   S704_BT_CODE_2018.RBT14_STANDARD_WELD_DATA := W#16#0;
   S704_BT_CODE_2018.RBT15_STANDARD_WELD_DATA := W#16#0;
   S704_BT_CODE_2018.RBT16_STANDARD_WELD_DATA := W#16#0;
   S704_BT_CODE_2018.RBT17_STANDARD_WELD_DATA := W#16#0;
   S704_BT_CODE_2018.RBT18_STANDARD_WELD_DATA := W#16#0;
   S704_BT_CODE_2018.RBT19_STANDARD_WELD_DATA := W#16#0;
   S704_BT_CODE_2018.RBT20_STANDARD_WELD_DATA := W#16#0;
   S704_BT_CODE_2018.RBT21_STANDARD_WELD_DATA := W#16#0;
   S704_BT_CODE_2018.RBT22_STANDARD_WELD_DATA := W#16#0;
   S704_BT_CODE_2018.RBT23_STANDARD_WELD_DAT := W#16#0;
   S704_BT_CODE_2018.RBT24_STANDARD_WELD_DAT := W#16#0;
   S704_BT_CODE_2018.CHK_WORD := W#16#0;
   S704_BT_CODE_2018.TEST_TEMP[1] := B#16#0;
   S704_BT_CODE_2018.TEST_TEMP[2] := B#16#0;
   S704_BT_CODE_2018.TEST_TEMP[3] := B#16#0;
   S704_BT_CODE_2018.TEST_TEMP[4] := B#16#0;
   S704_BT_CODE_2018.TEST_TEMP[5] := B#16#0;
   S704_BT_CODE_2018.TEST_TEMP[6] := B#16#0;
   S704_BT_CODE_2018.TEST_TEMP[7] := B#16#0;
   S704_BT_CODE_2018.TEST_TEMP[8] := B#16#0;
   S704_BT_CODE_2018.TEST_TEMP[9] := B#16#0;
   S704_BT_CODE_2018.TEST_TEMP[10] := B#16#0;
   S704_BT_CODE_2018.TEST_TEMP[11] := B#16#0;
   S704_BT_CODE_2018.TEST_TEMP[12] := B#16#0;
   S704_BT_CODE_2018.TEST_TEMP[13] := B#16#0;
   S704_BT_CODE_2018.TEST_TEMP[14] := B#16#0;
   S704_BT_CODE_2018.TEST_TEMP[15] := B#16#0;
   S704_BT_CODE_2018.TEST_TEMP[16] := B#16#0;
   S704_BT_CODE_2018.TEST_TEMP[17] := B#16#0;
   S704_BT_CODE_2018.TEST_TEMP[18] := B#16#0;
   S704_BT_CODE_2018.TEST_TEMP[19] := B#16#0;
   S704_BT_CODE_2018.TEST_TEMP[20] := B#16#0;
   S704_BT_CODE_2018.TEST_TEMP[21] := B#16#0;
   S704_BT_CODE_2018.TEST_TEMP[22] := B#16#0;
   S704_BT_CODE_2018.TEST_TEMP[23] := B#16#0;
   S704_BT_CODE_2018.TEST_TEMP[24] := B#16#0;
   S704_BT_CODE_2018.TEST_TEMP[25] := B#16#0;
   S704_BT_CODE_2018.TEST_TEMP[26] := B#16#0;
   S704_BT_CODE_2018.TEST_TEMP[27] := B#16#0;
   S704_BT_CODE_2018.TEST_TEMP[28] := B#16#0;
   S704_BT_CODE_2018.TEST_TEMP[29] := B#16#0;
   S704_BT_CODE_2018.TEST_TEMP[30] := B#16#0;
   S704_BT_CODE_2018.TEST_TEMP[31] := B#16#0;
   S704_BT_CODE_2018.TEST_TEMP[32] := B#16#0;
   S704_BT_CODE_2018.TEST_TEMP[33] := B#16#0;
   S704_BT_CODE_2018.TEST_TEMP[34] := B#16#0;
   S704_BT_CODE_2018.TEST_TEMP[35] := B#16#0;
   S704_BT_CODE_2018.TEST_TEMP[36] := B#16#0;
   S704_BT_CODE_2018.TEST_TEMP[37] := B#16#0;
   S704_BT_CODE_2018.TEST_TEMP[38] := B#16#0;
   S704_BT_CODE_2018.TEST_TEMP[39] := B#16#0;
   S704_BT_CODE_2018.TEST_TEMP[40] := B#16#0;
   S704_BT_CODE_2019.STATION_MAIN := W#16#0;
   S704_BT_CODE_2019.DISTINCTION_LH_RH := W#16#0;
   S704_BT_CODE_2019.STAION_NUMBER := W#16#0;
   S704_BT_CODE_2019.BODY_TYPE_1ST := W#16#0;
   S704_BT_CODE_2019.BODY_TYPE_OPTION := W#16#0;
   S704_BT_CODE_2019.RBT1_STANDARD_WELD_DATA := W#16#0;
   S704_BT_CODE_2019.RBT2_STANDARD_WELD_DATA := W#16#0;
   S704_BT_CODE_2019.RBT3_STANDARD_WELD_DATA := W#16#0;
   S704_BT_CODE_2019.RBT4_STANDARD_WELD_DATA := W#16#0;
   S704_BT_CODE_2019.RBT5_STANDARD_WELD_DATA := W#16#0;
   S704_BT_CODE_2019.RBT6_STANDARD_WELD_DATA := W#16#0;
   S704_BT_CODE_2019.RBT7_STANDARD_WELD_DATA := W#16#0;
   S704_BT_CODE_2019.RBT8_STANDARD_WELD_DATA := W#16#0;
   S704_BT_CODE_2019.RBT9_STANDARD_WELD_DATA := W#16#0;
   S704_BT_CODE_2019.RBT10_STANDARD_WELD_DATA := W#16#0;
   S704_BT_CODE_2019.RBT11_STANDARD_WELD_DATA := W#16#0;
   S704_BT_CODE_2019.RBT12_STANDARD_WELD_DATA := W#16#0;
   S704_BT_CODE_2019.RBT13_STANDARD_WELD_DATA := W#16#0;
   S704_BT_CODE_2019.RBT14_STANDARD_WELD_DATA := W#16#0;
   S704_BT_CODE_2019.RBT15_STANDARD_WELD_DATA := W#16#0;
   S704_BT_CODE_2019.RBT16_STANDARD_WELD_DATA := W#16#0;
   S704_BT_CODE_2019.RBT17_STANDARD_WELD_DATA := W#16#0;
   S704_BT_CODE_2019.RBT18_STANDARD_WELD_DATA := W#16#0;
   S704_BT_CODE_2019.RBT19_STANDARD_WELD_DATA := W#16#0;
   S704_BT_CODE_2019.RBT20_STANDARD_WELD_DATA := W#16#0;
   S704_BT_CODE_2019.RBT21_STANDARD_WELD_DATA := W#16#0;
   S704_BT_CODE_2019.RBT22_STANDARD_WELD_DATA := W#16#0;
   S704_BT_CODE_2019.RBT23_STANDARD_WELD_DAT := W#16#0;
   S704_BT_CODE_2019.RBT24_STANDARD_WELD_DAT := W#16#0;
   S704_BT_CODE_2019.CHK_WORD := W#16#0;
   S704_BT_CODE_2019.TEST_TEMP[1] := B#16#0;
   S704_BT_CODE_2019.TEST_TEMP[2] := B#16#0;
   S704_BT_CODE_2019.TEST_TEMP[3] := B#16#0;
   S704_BT_CODE_2019.TEST_TEMP[4] := B#16#0;
   S704_BT_CODE_2019.TEST_TEMP[5] := B#16#0;
   S704_BT_CODE_2019.TEST_TEMP[6] := B#16#0;
   S704_BT_CODE_2019.TEST_TEMP[7] := B#16#0;
   S704_BT_CODE_2019.TEST_TEMP[8] := B#16#0;
   S704_BT_CODE_2019.TEST_TEMP[9] := B#16#0;
   S704_BT_CODE_2019.TEST_TEMP[10] := B#16#0;
   S704_BT_CODE_2019.TEST_TEMP[11] := B#16#0;
   S704_BT_CODE_2019.TEST_TEMP[12] := B#16#0;
   S704_BT_CODE_2019.TEST_TEMP[13] := B#16#0;
   S704_BT_CODE_2019.TEST_TEMP[14] := B#16#0;
   S704_BT_CODE_2019.TEST_TEMP[15] := B#16#0;
   S704_BT_CODE_2019.TEST_TEMP[16] := B#16#0;
   S704_BT_CODE_2019.TEST_TEMP[17] := B#16#0;
   S704_BT_CODE_2019.TEST_TEMP[18] := B#16#0;
   S704_BT_CODE_2019.TEST_TEMP[19] := B#16#0;
   S704_BT_CODE_2019.TEST_TEMP[20] := B#16#0;
   S704_BT_CODE_2019.TEST_TEMP[21] := B#16#0;
   S704_BT_CODE_2019.TEST_TEMP[22] := B#16#0;
   S704_BT_CODE_2019.TEST_TEMP[23] := B#16#0;
   S704_BT_CODE_2019.TEST_TEMP[24] := B#16#0;
   S704_BT_CODE_2019.TEST_TEMP[25] := B#16#0;
   S704_BT_CODE_2019.TEST_TEMP[26] := B#16#0;
   S704_BT_CODE_2019.TEST_TEMP[27] := B#16#0;
   S704_BT_CODE_2019.TEST_TEMP[28] := B#16#0;
   S704_BT_CODE_2019.TEST_TEMP[29] := B#16#0;
   S704_BT_CODE_2019.TEST_TEMP[30] := B#16#0;
   S704_BT_CODE_2019.TEST_TEMP[31] := B#16#0;
   S704_BT_CODE_2019.TEST_TEMP[32] := B#16#0;
   S704_BT_CODE_2019.TEST_TEMP[33] := B#16#0;
   S704_BT_CODE_2019.TEST_TEMP[34] := B#16#0;
   S704_BT_CODE_2019.TEST_TEMP[35] := B#16#0;
   S704_BT_CODE_2019.TEST_TEMP[36] := B#16#0;
   S704_BT_CODE_2019.TEST_TEMP[37] := B#16#0;
   S704_BT_CODE_2019.TEST_TEMP[38] := B#16#0;
   S704_BT_CODE_2019.TEST_TEMP[39] := B#16#0;
   S704_BT_CODE_2019.TEST_TEMP[40] := B#16#0;
   S704_BT_CODE_2020.STATION_MAIN := W#16#0;
   S704_BT_CODE_2020.DISTINCTION_LH_RH := W#16#0;
   S704_BT_CODE_2020.STAION_NUMBER := W#16#0;
   S704_BT_CODE_2020.BODY_TYPE_1ST := W#16#0;
   S704_BT_CODE_2020.BODY_TYPE_OPTION := W#16#0;
   S704_BT_CODE_2020.RBT1_STANDARD_WELD_DATA := W#16#0;
   S704_BT_CODE_2020.RBT2_STANDARD_WELD_DATA := W#16#0;
   S704_BT_CODE_2020.RBT3_STANDARD_WELD_DATA := W#16#0;
   S704_BT_CODE_2020.RBT4_STANDARD_WELD_DATA := W#16#0;
   S704_BT_CODE_2020.RBT5_STANDARD_WELD_DATA := W#16#0;
   S704_BT_CODE_2020.RBT6_STANDARD_WELD_DATA := W#16#0;
   S704_BT_CODE_2020.RBT7_STANDARD_WELD_DATA := W#16#0;
   S704_BT_CODE_2020.RBT8_STANDARD_WELD_DATA := W#16#0;
   S704_BT_CODE_2020.RBT9_STANDARD_WELD_DATA := W#16#0;
   S704_BT_CODE_2020.RBT10_STANDARD_WELD_DATA := W#16#0;
   S704_BT_CODE_2020.RBT11_STANDARD_WELD_DATA := W#16#0;
   S704_BT_CODE_2020.RBT12_STANDARD_WELD_DATA := W#16#0;
   S704_BT_CODE_2020.RBT13_STANDARD_WELD_DATA := W#16#0;
   S704_BT_CODE_2020.RBT14_STANDARD_WELD_DATA := W#16#0;
   S704_BT_CODE_2020.RBT15_STANDARD_WELD_DATA := W#16#0;
   S704_BT_CODE_2020.RBT16_STANDARD_WELD_DATA := W#16#0;
   S704_BT_CODE_2020.RBT17_STANDARD_WELD_DATA := W#16#0;
   S704_BT_CODE_2020.RBT18_STANDARD_WELD_DATA := W#16#0;
   S704_BT_CODE_2020.RBT19_STANDARD_WELD_DATA := W#16#0;
   S704_BT_CODE_2020.RBT20_STANDARD_WELD_DATA := W#16#0;
   S704_BT_CODE_2020.RBT21_STANDARD_WELD_DATA := W#16#0;
   S704_BT_CODE_2020.RBT22_STANDARD_WELD_DATA := W#16#0;
   S704_BT_CODE_2020.RBT23_STANDARD_WELD_DAT := W#16#0;
   S704_BT_CODE_2020.RBT24_STANDARD_WELD_DAT := W#16#0;
   S704_BT_CODE_2020.CHK_WORD := W#16#0;
   S704_BT_CODE_2020.TEST_TEMP[1] := B#16#0;
   S704_BT_CODE_2020.TEST_TEMP[2] := B#16#0;
   S704_BT_CODE_2020.TEST_TEMP[3] := B#16#0;
   S704_BT_CODE_2020.TEST_TEMP[4] := B#16#0;
   S704_BT_CODE_2020.TEST_TEMP[5] := B#16#0;
   S704_BT_CODE_2020.TEST_TEMP[6] := B#16#0;
   S704_BT_CODE_2020.TEST_TEMP[7] := B#16#0;
   S704_BT_CODE_2020.TEST_TEMP[8] := B#16#0;
   S704_BT_CODE_2020.TEST_TEMP[9] := B#16#0;
   S704_BT_CODE_2020.TEST_TEMP[10] := B#16#0;
   S704_BT_CODE_2020.TEST_TEMP[11] := B#16#0;
   S704_BT_CODE_2020.TEST_TEMP[12] := B#16#0;
   S704_BT_CODE_2020.TEST_TEMP[13] := B#16#0;
   S704_BT_CODE_2020.TEST_TEMP[14] := B#16#0;
   S704_BT_CODE_2020.TEST_TEMP[15] := B#16#0;
   S704_BT_CODE_2020.TEST_TEMP[16] := B#16#0;
   S704_BT_CODE_2020.TEST_TEMP[17] := B#16#0;
   S704_BT_CODE_2020.TEST_TEMP[18] := B#16#0;
   S704_BT_CODE_2020.TEST_TEMP[19] := B#16#0;
   S704_BT_CODE_2020.TEST_TEMP[20] := B#16#0;
   S704_BT_CODE_2020.TEST_TEMP[21] := B#16#0;
   S704_BT_CODE_2020.TEST_TEMP[22] := B#16#0;
   S704_BT_CODE_2020.TEST_TEMP[23] := B#16#0;
   S704_BT_CODE_2020.TEST_TEMP[24] := B#16#0;
   S704_BT_CODE_2020.TEST_TEMP[25] := B#16#0;
   S704_BT_CODE_2020.TEST_TEMP[26] := B#16#0;
   S704_BT_CODE_2020.TEST_TEMP[27] := B#16#0;
   S704_BT_CODE_2020.TEST_TEMP[28] := B#16#0;
   S704_BT_CODE_2020.TEST_TEMP[29] := B#16#0;
   S704_BT_CODE_2020.TEST_TEMP[30] := B#16#0;
   S704_BT_CODE_2020.TEST_TEMP[31] := B#16#0;
   S704_BT_CODE_2020.TEST_TEMP[32] := B#16#0;
   S704_BT_CODE_2020.TEST_TEMP[33] := B#16#0;
   S704_BT_CODE_2020.TEST_TEMP[34] := B#16#0;
   S704_BT_CODE_2020.TEST_TEMP[35] := B#16#0;
   S704_BT_CODE_2020.TEST_TEMP[36] := B#16#0;
   S704_BT_CODE_2020.TEST_TEMP[37] := B#16#0;
   S704_BT_CODE_2020.TEST_TEMP[38] := B#16#0;
   S704_BT_CODE_2020.TEST_TEMP[39] := B#16#0;
   S704_BT_CODE_2020.TEST_TEMP[40] := B#16#0;
   S704_BT_CODE_2021.STATION_MAIN := W#16#0;
   S704_BT_CODE_2021.DISTINCTION_LH_RH := W#16#0;
   S704_BT_CODE_2021.STAION_NUMBER := W#16#0;
   S704_BT_CODE_2021.BODY_TYPE_1ST := W#16#0;
   S704_BT_CODE_2021.BODY_TYPE_OPTION := W#16#0;
   S704_BT_CODE_2021.RBT1_STANDARD_WELD_DATA := W#16#0;
   S704_BT_CODE_2021.RBT2_STANDARD_WELD_DATA := W#16#0;
   S704_BT_CODE_2021.RBT3_STANDARD_WELD_DATA := W#16#0;
   S704_BT_CODE_2021.RBT4_STANDARD_WELD_DATA := W#16#0;
   S704_BT_CODE_2021.RBT5_STANDARD_WELD_DATA := W#16#0;
   S704_BT_CODE_2021.RBT6_STANDARD_WELD_DATA := W#16#0;
   S704_BT_CODE_2021.RBT7_STANDARD_WELD_DATA := W#16#0;
   S704_BT_CODE_2021.RBT8_STANDARD_WELD_DATA := W#16#0;
   S704_BT_CODE_2021.RBT9_STANDARD_WELD_DATA := W#16#0;
   S704_BT_CODE_2021.RBT10_STANDARD_WELD_DATA := W#16#0;
   S704_BT_CODE_2021.RBT11_STANDARD_WELD_DATA := W#16#0;
   S704_BT_CODE_2021.RBT12_STANDARD_WELD_DATA := W#16#0;
   S704_BT_CODE_2021.RBT13_STANDARD_WELD_DATA := W#16#0;
   S704_BT_CODE_2021.RBT14_STANDARD_WELD_DATA := W#16#0;
   S704_BT_CODE_2021.RBT15_STANDARD_WELD_DATA := W#16#0;
   S704_BT_CODE_2021.RBT16_STANDARD_WELD_DATA := W#16#0;
   S704_BT_CODE_2021.RBT17_STANDARD_WELD_DATA := W#16#0;
   S704_BT_CODE_2021.RBT18_STANDARD_WELD_DATA := W#16#0;
   S704_BT_CODE_2021.RBT19_STANDARD_WELD_DATA := W#16#0;
   S704_BT_CODE_2021.RBT20_STANDARD_WELD_DATA := W#16#0;
   S704_BT_CODE_2021.RBT21_STANDARD_WELD_DATA := W#16#0;
   S704_BT_CODE_2021.RBT22_STANDARD_WELD_DATA := W#16#0;
   S704_BT_CODE_2021.RBT23_STANDARD_WELD_DAT := W#16#0;
   S704_BT_CODE_2021.RBT24_STANDARD_WELD_DAT := W#16#0;
   S704_BT_CODE_2021.CHK_WORD := W#16#0;
   S704_BT_CODE_2021.TEST_TEMP[1] := B#16#0;
   S704_BT_CODE_2021.TEST_TEMP[2] := B#16#0;
   S704_BT_CODE_2021.TEST_TEMP[3] := B#16#0;
   S704_BT_CODE_2021.TEST_TEMP[4] := B#16#0;
   S704_BT_CODE_2021.TEST_TEMP[5] := B#16#0;
   S704_BT_CODE_2021.TEST_TEMP[6] := B#16#0;
   S704_BT_CODE_2021.TEST_TEMP[7] := B#16#0;
   S704_BT_CODE_2021.TEST_TEMP[8] := B#16#0;
   S704_BT_CODE_2021.TEST_TEMP[9] := B#16#0;
   S704_BT_CODE_2021.TEST_TEMP[10] := B#16#0;
   S704_BT_CODE_2021.TEST_TEMP[11] := B#16#0;
   S704_BT_CODE_2021.TEST_TEMP[12] := B#16#0;
   S704_BT_CODE_2021.TEST_TEMP[13] := B#16#0;
   S704_BT_CODE_2021.TEST_TEMP[14] := B#16#0;
   S704_BT_CODE_2021.TEST_TEMP[15] := B#16#0;
   S704_BT_CODE_2021.TEST_TEMP[16] := B#16#0;
   S704_BT_CODE_2021.TEST_TEMP[17] := B#16#0;
   S704_BT_CODE_2021.TEST_TEMP[18] := B#16#0;
   S704_BT_CODE_2021.TEST_TEMP[19] := B#16#0;
   S704_BT_CODE_2021.TEST_TEMP[20] := B#16#0;
   S704_BT_CODE_2021.TEST_TEMP[21] := B#16#0;
   S704_BT_CODE_2021.TEST_TEMP[22] := B#16#0;
   S704_BT_CODE_2021.TEST_TEMP[23] := B#16#0;
   S704_BT_CODE_2021.TEST_TEMP[24] := B#16#0;
   S704_BT_CODE_2021.TEST_TEMP[25] := B#16#0;
   S704_BT_CODE_2021.TEST_TEMP[26] := B#16#0;
   S704_BT_CODE_2021.TEST_TEMP[27] := B#16#0;
   S704_BT_CODE_2021.TEST_TEMP[28] := B#16#0;
   S704_BT_CODE_2021.TEST_TEMP[29] := B#16#0;
   S704_BT_CODE_2021.TEST_TEMP[30] := B#16#0;
   S704_BT_CODE_2021.TEST_TEMP[31] := B#16#0;
   S704_BT_CODE_2021.TEST_TEMP[32] := B#16#0;
   S704_BT_CODE_2021.TEST_TEMP[33] := B#16#0;
   S704_BT_CODE_2021.TEST_TEMP[34] := B#16#0;
   S704_BT_CODE_2021.TEST_TEMP[35] := B#16#0;
   S704_BT_CODE_2021.TEST_TEMP[36] := B#16#0;
   S704_BT_CODE_2021.TEST_TEMP[37] := B#16#0;
   S704_BT_CODE_2021.TEST_TEMP[38] := B#16#0;
   S704_BT_CODE_2021.TEST_TEMP[39] := B#16#0;
   S704_BT_CODE_2021.TEST_TEMP[40] := B#16#0;
   S704_BT_CODE_2022.STATION_MAIN := W#16#0;
   S704_BT_CODE_2022.DISTINCTION_LH_RH := W#16#0;
   S704_BT_CODE_2022.STAION_NUMBER := W#16#0;
   S704_BT_CODE_2022.BODY_TYPE_1ST := W#16#0;
   S704_BT_CODE_2022.BODY_TYPE_OPTION := W#16#0;
   S704_BT_CODE_2022.RBT1_STANDARD_WELD_DATA := W#16#0;
   S704_BT_CODE_2022.RBT2_STANDARD_WELD_DATA := W#16#0;
   S704_BT_CODE_2022.RBT3_STANDARD_WELD_DATA := W#16#0;
   S704_BT_CODE_2022.RBT4_STANDARD_WELD_DATA := W#16#0;
   S704_BT_CODE_2022.RBT5_STANDARD_WELD_DATA := W#16#0;
   S704_BT_CODE_2022.RBT6_STANDARD_WELD_DATA := W#16#0;
   S704_BT_CODE_2022.RBT7_STANDARD_WELD_DATA := W#16#0;
   S704_BT_CODE_2022.RBT8_STANDARD_WELD_DATA := W#16#0;
   S704_BT_CODE_2022.RBT9_STANDARD_WELD_DATA := W#16#0;
   S704_BT_CODE_2022.RBT10_STANDARD_WELD_DATA := W#16#0;
   S704_BT_CODE_2022.RBT11_STANDARD_WELD_DATA := W#16#0;
   S704_BT_CODE_2022.RBT12_STANDARD_WELD_DATA := W#16#0;
   S704_BT_CODE_2022.RBT13_STANDARD_WELD_DATA := W#16#0;
   S704_BT_CODE_2022.RBT14_STANDARD_WELD_DATA := W#16#0;
   S704_BT_CODE_2022.RBT15_STANDARD_WELD_DATA := W#16#0;
   S704_BT_CODE_2022.RBT16_STANDARD_WELD_DATA := W#16#0;
   S704_BT_CODE_2022.RBT17_STANDARD_WELD_DATA := W#16#0;
   S704_BT_CODE_2022.RBT18_STANDARD_WELD_DATA := W#16#0;
   S704_BT_CODE_2022.RBT19_STANDARD_WELD_DATA := W#16#0;
   S704_BT_CODE_2022.RBT20_STANDARD_WELD_DATA := W#16#0;
   S704_BT_CODE_2022.RBT21_STANDARD_WELD_DATA := W#16#0;
   S704_BT_CODE_2022.RBT22_STANDARD_WELD_DATA := W#16#0;
   S704_BT_CODE_2022.RBT23_STANDARD_WELD_DAT := W#16#0;
   S704_BT_CODE_2022.RBT24_STANDARD_WELD_DAT := W#16#0;
   S704_BT_CODE_2022.CHK_WORD := W#16#0;
   S704_BT_CODE_2022.TEST_TEMP[1] := B#16#0;
   S704_BT_CODE_2022.TEST_TEMP[2] := B#16#0;
   S704_BT_CODE_2022.TEST_TEMP[3] := B#16#0;
   S704_BT_CODE_2022.TEST_TEMP[4] := B#16#0;
   S704_BT_CODE_2022.TEST_TEMP[5] := B#16#0;
   S704_BT_CODE_2022.TEST_TEMP[6] := B#16#0;
   S704_BT_CODE_2022.TEST_TEMP[7] := B#16#0;
   S704_BT_CODE_2022.TEST_TEMP[8] := B#16#0;
   S704_BT_CODE_2022.TEST_TEMP[9] := B#16#0;
   S704_BT_CODE_2022.TEST_TEMP[10] := B#16#0;
   S704_BT_CODE_2022.TEST_TEMP[11] := B#16#0;
   S704_BT_CODE_2022.TEST_TEMP[12] := B#16#0;
   S704_BT_CODE_2022.TEST_TEMP[13] := B#16#0;
   S704_BT_CODE_2022.TEST_TEMP[14] := B#16#0;
   S704_BT_CODE_2022.TEST_TEMP[15] := B#16#0;
   S704_BT_CODE_2022.TEST_TEMP[16] := B#16#0;
   S704_BT_CODE_2022.TEST_TEMP[17] := B#16#0;
   S704_BT_CODE_2022.TEST_TEMP[18] := B#16#0;
   S704_BT_CODE_2022.TEST_TEMP[19] := B#16#0;
   S704_BT_CODE_2022.TEST_TEMP[20] := B#16#0;
   S704_BT_CODE_2022.TEST_TEMP[21] := B#16#0;
   S704_BT_CODE_2022.TEST_TEMP[22] := B#16#0;
   S704_BT_CODE_2022.TEST_TEMP[23] := B#16#0;
   S704_BT_CODE_2022.TEST_TEMP[24] := B#16#0;
   S704_BT_CODE_2022.TEST_TEMP[25] := B#16#0;
   S704_BT_CODE_2022.TEST_TEMP[26] := B#16#0;
   S704_BT_CODE_2022.TEST_TEMP[27] := B#16#0;
   S704_BT_CODE_2022.TEST_TEMP[28] := B#16#0;
   S704_BT_CODE_2022.TEST_TEMP[29] := B#16#0;
   S704_BT_CODE_2022.TEST_TEMP[30] := B#16#0;
   S704_BT_CODE_2022.TEST_TEMP[31] := B#16#0;
   S704_BT_CODE_2022.TEST_TEMP[32] := B#16#0;
   S704_BT_CODE_2022.TEST_TEMP[33] := B#16#0;
   S704_BT_CODE_2022.TEST_TEMP[34] := B#16#0;
   S704_BT_CODE_2022.TEST_TEMP[35] := B#16#0;
   S704_BT_CODE_2022.TEST_TEMP[36] := B#16#0;
   S704_BT_CODE_2022.TEST_TEMP[37] := B#16#0;
   S704_BT_CODE_2022.TEST_TEMP[38] := B#16#0;
   S704_BT_CODE_2022.TEST_TEMP[39] := B#16#0;
   S704_BT_CODE_2022.TEST_TEMP[40] := B#16#0;
   S704_BT_CODE_2023.STATION_MAIN := W#16#0;
   S704_BT_CODE_2023.DISTINCTION_LH_RH := W#16#0;
   S704_BT_CODE_2023.STAION_NUMBER := W#16#0;
   S704_BT_CODE_2023.BODY_TYPE_1ST := W#16#0;
   S704_BT_CODE_2023.BODY_TYPE_OPTION := W#16#0;
   S704_BT_CODE_2023.RBT1_STANDARD_WELD_DATA := W#16#0;
   S704_BT_CODE_2023.RBT2_STANDARD_WELD_DATA := W#16#0;
   S704_BT_CODE_2023.RBT3_STANDARD_WELD_DATA := W#16#0;
   S704_BT_CODE_2023.RBT4_STANDARD_WELD_DATA := W#16#0;
   S704_BT_CODE_2023.RBT5_STANDARD_WELD_DATA := W#16#0;
   S704_BT_CODE_2023.RBT6_STANDARD_WELD_DATA := W#16#0;
   S704_BT_CODE_2023.RBT7_STANDARD_WELD_DATA := W#16#0;
   S704_BT_CODE_2023.RBT8_STANDARD_WELD_DATA := W#16#0;
   S704_BT_CODE_2023.RBT9_STANDARD_WELD_DATA := W#16#0;
   S704_BT_CODE_2023.RBT10_STANDARD_WELD_DATA := W#16#0;
   S704_BT_CODE_2023.RBT11_STANDARD_WELD_DATA := W#16#0;
   S704_BT_CODE_2023.RBT12_STANDARD_WELD_DATA := W#16#0;
   S704_BT_CODE_2023.RBT13_STANDARD_WELD_DATA := W#16#0;
   S704_BT_CODE_2023.RBT14_STANDARD_WELD_DATA := W#16#0;
   S704_BT_CODE_2023.RBT15_STANDARD_WELD_DATA := W#16#0;
   S704_BT_CODE_2023.RBT16_STANDARD_WELD_DATA := W#16#0;
   S704_BT_CODE_2023.RBT17_STANDARD_WELD_DATA := W#16#0;
   S704_BT_CODE_2023.RBT18_STANDARD_WELD_DATA := W#16#0;
   S704_BT_CODE_2023.RBT19_STANDARD_WELD_DATA := W#16#0;
   S704_BT_CODE_2023.RBT20_STANDARD_WELD_DATA := W#16#0;
   S704_BT_CODE_2023.RBT21_STANDARD_WELD_DATA := W#16#0;
   S704_BT_CODE_2023.RBT22_STANDARD_WELD_DATA := W#16#0;
   S704_BT_CODE_2023.RBT23_STANDARD_WELD_DAT := W#16#0;
   S704_BT_CODE_2023.RBT24_STANDARD_WELD_DAT := W#16#0;
   S704_BT_CODE_2023.CHK_WORD := W#16#0;
   S704_BT_CODE_2023.TEST_TEMP[1] := B#16#0;
   S704_BT_CODE_2023.TEST_TEMP[2] := B#16#0;
   S704_BT_CODE_2023.TEST_TEMP[3] := B#16#0;
   S704_BT_CODE_2023.TEST_TEMP[4] := B#16#0;
   S704_BT_CODE_2023.TEST_TEMP[5] := B#16#0;
   S704_BT_CODE_2023.TEST_TEMP[6] := B#16#0;
   S704_BT_CODE_2023.TEST_TEMP[7] := B#16#0;
   S704_BT_CODE_2023.TEST_TEMP[8] := B#16#0;
   S704_BT_CODE_2023.TEST_TEMP[9] := B#16#0;
   S704_BT_CODE_2023.TEST_TEMP[10] := B#16#0;
   S704_BT_CODE_2023.TEST_TEMP[11] := B#16#0;
   S704_BT_CODE_2023.TEST_TEMP[12] := B#16#0;
   S704_BT_CODE_2023.TEST_TEMP[13] := B#16#0;
   S704_BT_CODE_2023.TEST_TEMP[14] := B#16#0;
   S704_BT_CODE_2023.TEST_TEMP[15] := B#16#0;
   S704_BT_CODE_2023.TEST_TEMP[16] := B#16#0;
   S704_BT_CODE_2023.TEST_TEMP[17] := B#16#0;
   S704_BT_CODE_2023.TEST_TEMP[18] := B#16#0;
   S704_BT_CODE_2023.TEST_TEMP[19] := B#16#0;
   S704_BT_CODE_2023.TEST_TEMP[20] := B#16#0;
   S704_BT_CODE_2023.TEST_TEMP[21] := B#16#0;
   S704_BT_CODE_2023.TEST_TEMP[22] := B#16#0;
   S704_BT_CODE_2023.TEST_TEMP[23] := B#16#0;
   S704_BT_CODE_2023.TEST_TEMP[24] := B#16#0;
   S704_BT_CODE_2023.TEST_TEMP[25] := B#16#0;
   S704_BT_CODE_2023.TEST_TEMP[26] := B#16#0;
   S704_BT_CODE_2023.TEST_TEMP[27] := B#16#0;
   S704_BT_CODE_2023.TEST_TEMP[28] := B#16#0;
   S704_BT_CODE_2023.TEST_TEMP[29] := B#16#0;
   S704_BT_CODE_2023.TEST_TEMP[30] := B#16#0;
   S704_BT_CODE_2023.TEST_TEMP[31] := B#16#0;
   S704_BT_CODE_2023.TEST_TEMP[32] := B#16#0;
   S704_BT_CODE_2023.TEST_TEMP[33] := B#16#0;
   S704_BT_CODE_2023.TEST_TEMP[34] := B#16#0;
   S704_BT_CODE_2023.TEST_TEMP[35] := B#16#0;
   S704_BT_CODE_2023.TEST_TEMP[36] := B#16#0;
   S704_BT_CODE_2023.TEST_TEMP[37] := B#16#0;
   S704_BT_CODE_2023.TEST_TEMP[38] := B#16#0;
   S704_BT_CODE_2023.TEST_TEMP[39] := B#16#0;
   S704_BT_CODE_2023.TEST_TEMP[40] := B#16#0;
   S704_BT_CODE_2024.STATION_MAIN := W#16#0;
   S704_BT_CODE_2024.DISTINCTION_LH_RH := W#16#0;
   S704_BT_CODE_2024.STAION_NUMBER := W#16#0;
   S704_BT_CODE_2024.BODY_TYPE_1ST := W#16#0;
   S704_BT_CODE_2024.BODY_TYPE_OPTION := W#16#0;
   S704_BT_CODE_2024.RBT1_STANDARD_WELD_DATA := W#16#0;
   S704_BT_CODE_2024.RBT2_STANDARD_WELD_DATA := W#16#0;
   S704_BT_CODE_2024.RBT3_STANDARD_WELD_DATA := W#16#0;
   S704_BT_CODE_2024.RBT4_STANDARD_WELD_DATA := W#16#0;
   S704_BT_CODE_2024.RBT5_STANDARD_WELD_DATA := W#16#0;
   S704_BT_CODE_2024.RBT6_STANDARD_WELD_DATA := W#16#0;
   S704_BT_CODE_2024.RBT7_STANDARD_WELD_DATA := W#16#0;
   S704_BT_CODE_2024.RBT8_STANDARD_WELD_DATA := W#16#0;
   S704_BT_CODE_2024.RBT9_STANDARD_WELD_DATA := W#16#0;
   S704_BT_CODE_2024.RBT10_STANDARD_WELD_DATA := W#16#0;
   S704_BT_CODE_2024.RBT11_STANDARD_WELD_DATA := W#16#0;
   S704_BT_CODE_2024.RBT12_STANDARD_WELD_DATA := W#16#0;
   S704_BT_CODE_2024.RBT13_STANDARD_WELD_DATA := W#16#0;
   S704_BT_CODE_2024.RBT14_STANDARD_WELD_DATA := W#16#0;
   S704_BT_CODE_2024.RBT15_STANDARD_WELD_DATA := W#16#0;
   S704_BT_CODE_2024.RBT16_STANDARD_WELD_DATA := W#16#0;
   S704_BT_CODE_2024.RBT17_STANDARD_WELD_DATA := W#16#0;
   S704_BT_CODE_2024.RBT18_STANDARD_WELD_DATA := W#16#0;
   S704_BT_CODE_2024.RBT19_STANDARD_WELD_DATA := W#16#0;
   S704_BT_CODE_2024.RBT20_STANDARD_WELD_DATA := W#16#0;
   S704_BT_CODE_2024.RBT21_STANDARD_WELD_DATA := W#16#0;
   S704_BT_CODE_2024.RBT22_STANDARD_WELD_DATA := W#16#0;
   S704_BT_CODE_2024.RBT23_STANDARD_WELD_DAT := W#16#0;
   S704_BT_CODE_2024.RBT24_STANDARD_WELD_DAT := W#16#0;
   S704_BT_CODE_2024.CHK_WORD := W#16#0;
   S704_BT_CODE_2024.TEST_TEMP[1] := B#16#0;
   S704_BT_CODE_2024.TEST_TEMP[2] := B#16#0;
   S704_BT_CODE_2024.TEST_TEMP[3] := B#16#0;
   S704_BT_CODE_2024.TEST_TEMP[4] := B#16#0;
   S704_BT_CODE_2024.TEST_TEMP[5] := B#16#0;
   S704_BT_CODE_2024.TEST_TEMP[6] := B#16#0;
   S704_BT_CODE_2024.TEST_TEMP[7] := B#16#0;
   S704_BT_CODE_2024.TEST_TEMP[8] := B#16#0;
   S704_BT_CODE_2024.TEST_TEMP[9] := B#16#0;
   S704_BT_CODE_2024.TEST_TEMP[10] := B#16#0;
   S704_BT_CODE_2024.TEST_TEMP[11] := B#16#0;
   S704_BT_CODE_2024.TEST_TEMP[12] := B#16#0;
   S704_BT_CODE_2024.TEST_TEMP[13] := B#16#0;
   S704_BT_CODE_2024.TEST_TEMP[14] := B#16#0;
   S704_BT_CODE_2024.TEST_TEMP[15] := B#16#0;
   S704_BT_CODE_2024.TEST_TEMP[16] := B#16#0;
   S704_BT_CODE_2024.TEST_TEMP[17] := B#16#0;
   S704_BT_CODE_2024.TEST_TEMP[18] := B#16#0;
   S704_BT_CODE_2024.TEST_TEMP[19] := B#16#0;
   S704_BT_CODE_2024.TEST_TEMP[20] := B#16#0;
   S704_BT_CODE_2024.TEST_TEMP[21] := B#16#0;
   S704_BT_CODE_2024.TEST_TEMP[22] := B#16#0;
   S704_BT_CODE_2024.TEST_TEMP[23] := B#16#0;
   S704_BT_CODE_2024.TEST_TEMP[24] := B#16#0;
   S704_BT_CODE_2024.TEST_TEMP[25] := B#16#0;
   S704_BT_CODE_2024.TEST_TEMP[26] := B#16#0;
   S704_BT_CODE_2024.TEST_TEMP[27] := B#16#0;
   S704_BT_CODE_2024.TEST_TEMP[28] := B#16#0;
   S704_BT_CODE_2024.TEST_TEMP[29] := B#16#0;
   S704_BT_CODE_2024.TEST_TEMP[30] := B#16#0;
   S704_BT_CODE_2024.TEST_TEMP[31] := B#16#0;
   S704_BT_CODE_2024.TEST_TEMP[32] := B#16#0;
   S704_BT_CODE_2024.TEST_TEMP[33] := B#16#0;
   S704_BT_CODE_2024.TEST_TEMP[34] := B#16#0;
   S704_BT_CODE_2024.TEST_TEMP[35] := B#16#0;
   S704_BT_CODE_2024.TEST_TEMP[36] := B#16#0;
   S704_BT_CODE_2024.TEST_TEMP[37] := B#16#0;
   S704_BT_CODE_2024.TEST_TEMP[38] := B#16#0;
   S704_BT_CODE_2024.TEST_TEMP[39] := B#16#0;
   S704_BT_CODE_2024.TEST_TEMP[40] := B#16#0;
   S704_BT_CODE_2025.STATION_MAIN := W#16#0;
   S704_BT_CODE_2025.DISTINCTION_LH_RH := W#16#0;
   S704_BT_CODE_2025.STAION_NUMBER := W#16#0;
   S704_BT_CODE_2025.BODY_TYPE_1ST := W#16#0;
   S704_BT_CODE_2025.BODY_TYPE_OPTION := W#16#0;
   S704_BT_CODE_2025.RBT1_STANDARD_WELD_DATA := W#16#0;
   S704_BT_CODE_2025.RBT2_STANDARD_WELD_DATA := W#16#0;
   S704_BT_CODE_2025.RBT3_STANDARD_WELD_DATA := W#16#0;
   S704_BT_CODE_2025.RBT4_STANDARD_WELD_DATA := W#16#0;
   S704_BT_CODE_2025.RBT5_STANDARD_WELD_DATA := W#16#0;
   S704_BT_CODE_2025.RBT6_STANDARD_WELD_DATA := W#16#0;
   S704_BT_CODE_2025.RBT7_STANDARD_WELD_DATA := W#16#0;
   S704_BT_CODE_2025.RBT8_STANDARD_WELD_DATA := W#16#0;
   S704_BT_CODE_2025.RBT9_STANDARD_WELD_DATA := W#16#0;
   S704_BT_CODE_2025.RBT10_STANDARD_WELD_DATA := W#16#0;
   S704_BT_CODE_2025.RBT11_STANDARD_WELD_DATA := W#16#0;
   S704_BT_CODE_2025.RBT12_STANDARD_WELD_DATA := W#16#0;
   S704_BT_CODE_2025.RBT13_STANDARD_WELD_DATA := W#16#0;
   S704_BT_CODE_2025.RBT14_STANDARD_WELD_DATA := W#16#0;
   S704_BT_CODE_2025.RBT15_STANDARD_WELD_DATA := W#16#0;
   S704_BT_CODE_2025.RBT16_STANDARD_WELD_DATA := W#16#0;
   S704_BT_CODE_2025.RBT17_STANDARD_WELD_DATA := W#16#0;
   S704_BT_CODE_2025.RBT18_STANDARD_WELD_DATA := W#16#0;
   S704_BT_CODE_2025.RBT19_STANDARD_WELD_DATA := W#16#0;
   S704_BT_CODE_2025.RBT20_STANDARD_WELD_DATA := W#16#0;
   S704_BT_CODE_2025.RBT21_STANDARD_WELD_DATA := W#16#0;
   S704_BT_CODE_2025.RBT22_STANDARD_WELD_DATA := W#16#0;
   S704_BT_CODE_2025.RBT23_STANDARD_WELD_DAT := W#16#0;
   S704_BT_CODE_2025.RBT24_STANDARD_WELD_DAT := W#16#0;
   S704_BT_CODE_2025.CHK_WORD := W#16#0;
   S704_BT_CODE_2025.TEST_TEMP[1] := B#16#0;
   S704_BT_CODE_2025.TEST_TEMP[2] := B#16#0;
   S704_BT_CODE_2025.TEST_TEMP[3] := B#16#0;
   S704_BT_CODE_2025.TEST_TEMP[4] := B#16#0;
   S704_BT_CODE_2025.TEST_TEMP[5] := B#16#0;
   S704_BT_CODE_2025.TEST_TEMP[6] := B#16#0;
   S704_BT_CODE_2025.TEST_TEMP[7] := B#16#0;
   S704_BT_CODE_2025.TEST_TEMP[8] := B#16#0;
   S704_BT_CODE_2025.TEST_TEMP[9] := B#16#0;
   S704_BT_CODE_2025.TEST_TEMP[10] := B#16#0;
   S704_BT_CODE_2025.TEST_TEMP[11] := B#16#0;
   S704_BT_CODE_2025.TEST_TEMP[12] := B#16#0;
   S704_BT_CODE_2025.TEST_TEMP[13] := B#16#0;
   S704_BT_CODE_2025.TEST_TEMP[14] := B#16#0;
   S704_BT_CODE_2025.TEST_TEMP[15] := B#16#0;
   S704_BT_CODE_2025.TEST_TEMP[16] := B#16#0;
   S704_BT_CODE_2025.TEST_TEMP[17] := B#16#0;
   S704_BT_CODE_2025.TEST_TEMP[18] := B#16#0;
   S704_BT_CODE_2025.TEST_TEMP[19] := B#16#0;
   S704_BT_CODE_2025.TEST_TEMP[20] := B#16#0;
   S704_BT_CODE_2025.TEST_TEMP[21] := B#16#0;
   S704_BT_CODE_2025.TEST_TEMP[22] := B#16#0;
   S704_BT_CODE_2025.TEST_TEMP[23] := B#16#0;
   S704_BT_CODE_2025.TEST_TEMP[24] := B#16#0;
   S704_BT_CODE_2025.TEST_TEMP[25] := B#16#0;
   S704_BT_CODE_2025.TEST_TEMP[26] := B#16#0;
   S704_BT_CODE_2025.TEST_TEMP[27] := B#16#0;
   S704_BT_CODE_2025.TEST_TEMP[28] := B#16#0;
   S704_BT_CODE_2025.TEST_TEMP[29] := B#16#0;
   S704_BT_CODE_2025.TEST_TEMP[30] := B#16#0;
   S704_BT_CODE_2025.TEST_TEMP[31] := B#16#0;
   S704_BT_CODE_2025.TEST_TEMP[32] := B#16#0;
   S704_BT_CODE_2025.TEST_TEMP[33] := B#16#0;
   S704_BT_CODE_2025.TEST_TEMP[34] := B#16#0;
   S704_BT_CODE_2025.TEST_TEMP[35] := B#16#0;
   S704_BT_CODE_2025.TEST_TEMP[36] := B#16#0;
   S704_BT_CODE_2025.TEST_TEMP[37] := B#16#0;
   S704_BT_CODE_2025.TEST_TEMP[38] := B#16#0;
   S704_BT_CODE_2025.TEST_TEMP[39] := B#16#0;
   S704_BT_CODE_2025.TEST_TEMP[40] := B#16#0;
   S704_BT_CODE_2026.STATION_MAIN := W#16#0;
   S704_BT_CODE_2026.DISTINCTION_LH_RH := W#16#0;
   S704_BT_CODE_2026.STAION_NUMBER := W#16#0;
   S704_BT_CODE_2026.BODY_TYPE_1ST := W#16#0;
   S704_BT_CODE_2026.BODY_TYPE_OPTION := W#16#0;
   S704_BT_CODE_2026.RBT1_STANDARD_WELD_DATA := W#16#0;
   S704_BT_CODE_2026.RBT2_STANDARD_WELD_DATA := W#16#0;
   S704_BT_CODE_2026.RBT3_STANDARD_WELD_DATA := W#16#0;
   S704_BT_CODE_2026.RBT4_STANDARD_WELD_DATA := W#16#0;
   S704_BT_CODE_2026.RBT5_STANDARD_WELD_DATA := W#16#0;
   S704_BT_CODE_2026.RBT6_STANDARD_WELD_DATA := W#16#0;
   S704_BT_CODE_2026.RBT7_STANDARD_WELD_DATA := W#16#0;
   S704_BT_CODE_2026.RBT8_STANDARD_WELD_DATA := W#16#0;
   S704_BT_CODE_2026.RBT9_STANDARD_WELD_DATA := W#16#0;
   S704_BT_CODE_2026.RBT10_STANDARD_WELD_DATA := W#16#0;
   S704_BT_CODE_2026.RBT11_STANDARD_WELD_DATA := W#16#0;
   S704_BT_CODE_2026.RBT12_STANDARD_WELD_DATA := W#16#0;
   S704_BT_CODE_2026.RBT13_STANDARD_WELD_DATA := W#16#0;
   S704_BT_CODE_2026.RBT14_STANDARD_WELD_DATA := W#16#0;
   S704_BT_CODE_2026.RBT15_STANDARD_WELD_DATA := W#16#0;
   S704_BT_CODE_2026.RBT16_STANDARD_WELD_DATA := W#16#0;
   S704_BT_CODE_2026.RBT17_STANDARD_WELD_DATA := W#16#0;
   S704_BT_CODE_2026.RBT18_STANDARD_WELD_DATA := W#16#0;
   S704_BT_CODE_2026.RBT19_STANDARD_WELD_DATA := W#16#0;
   S704_BT_CODE_2026.RBT20_STANDARD_WELD_DATA := W#16#0;
   S704_BT_CODE_2026.RBT21_STANDARD_WELD_DATA := W#16#0;
   S704_BT_CODE_2026.RBT22_STANDARD_WELD_DATA := W#16#0;
   S704_BT_CODE_2026.RBT23_STANDARD_WELD_DAT := W#16#0;
   S704_BT_CODE_2026.RBT24_STANDARD_WELD_DAT := W#16#0;
   S704_BT_CODE_2026.CHK_WORD := W#16#0;
   S704_BT_CODE_2026.TEST_TEMP[1] := B#16#0;
   S704_BT_CODE_2026.TEST_TEMP[2] := B#16#0;
   S704_BT_CODE_2026.TEST_TEMP[3] := B#16#0;
   S704_BT_CODE_2026.TEST_TEMP[4] := B#16#0;
   S704_BT_CODE_2026.TEST_TEMP[5] := B#16#0;
   S704_BT_CODE_2026.TEST_TEMP[6] := B#16#0;
   S704_BT_CODE_2026.TEST_TEMP[7] := B#16#0;
   S704_BT_CODE_2026.TEST_TEMP[8] := B#16#0;
   S704_BT_CODE_2026.TEST_TEMP[9] := B#16#0;
   S704_BT_CODE_2026.TEST_TEMP[10] := B#16#0;
   S704_BT_CODE_2026.TEST_TEMP[11] := B#16#0;
   S704_BT_CODE_2026.TEST_TEMP[12] := B#16#0;
   S704_BT_CODE_2026.TEST_TEMP[13] := B#16#0;
   S704_BT_CODE_2026.TEST_TEMP[14] := B#16#0;
   S704_BT_CODE_2026.TEST_TEMP[15] := B#16#0;
   S704_BT_CODE_2026.TEST_TEMP[16] := B#16#0;
   S704_BT_CODE_2026.TEST_TEMP[17] := B#16#0;
   S704_BT_CODE_2026.TEST_TEMP[18] := B#16#0;
   S704_BT_CODE_2026.TEST_TEMP[19] := B#16#0;
   S704_BT_CODE_2026.TEST_TEMP[20] := B#16#0;
   S704_BT_CODE_2026.TEST_TEMP[21] := B#16#0;
   S704_BT_CODE_2026.TEST_TEMP[22] := B#16#0;
   S704_BT_CODE_2026.TEST_TEMP[23] := B#16#0;
   S704_BT_CODE_2026.TEST_TEMP[24] := B#16#0;
   S704_BT_CODE_2026.TEST_TEMP[25] := B#16#0;
   S704_BT_CODE_2026.TEST_TEMP[26] := B#16#0;
   S704_BT_CODE_2026.TEST_TEMP[27] := B#16#0;
   S704_BT_CODE_2026.TEST_TEMP[28] := B#16#0;
   S704_BT_CODE_2026.TEST_TEMP[29] := B#16#0;
   S704_BT_CODE_2026.TEST_TEMP[30] := B#16#0;
   S704_BT_CODE_2026.TEST_TEMP[31] := B#16#0;
   S704_BT_CODE_2026.TEST_TEMP[32] := B#16#0;
   S704_BT_CODE_2026.TEST_TEMP[33] := B#16#0;
   S704_BT_CODE_2026.TEST_TEMP[34] := B#16#0;
   S704_BT_CODE_2026.TEST_TEMP[35] := B#16#0;
   S704_BT_CODE_2026.TEST_TEMP[36] := B#16#0;
   S704_BT_CODE_2026.TEST_TEMP[37] := B#16#0;
   S704_BT_CODE_2026.TEST_TEMP[38] := B#16#0;
   S704_BT_CODE_2026.TEST_TEMP[39] := B#16#0;
   S704_BT_CODE_2026.TEST_TEMP[40] := B#16#0;
   S704_BT_CODE_2027.STATION_MAIN := W#16#0;
   S704_BT_CODE_2027.DISTINCTION_LH_RH := W#16#0;
   S704_BT_CODE_2027.STAION_NUMBER := W#16#0;
   S704_BT_CODE_2027.BODY_TYPE_1ST := W#16#0;
   S704_BT_CODE_2027.BODY_TYPE_OPTION := W#16#0;
   S704_BT_CODE_2027.RBT1_STANDARD_WELD_DATA := W#16#0;
   S704_BT_CODE_2027.RBT2_STANDARD_WELD_DATA := W#16#0;
   S704_BT_CODE_2027.RBT3_STANDARD_WELD_DATA := W#16#0;
   S704_BT_CODE_2027.RBT4_STANDARD_WELD_DATA := W#16#0;
   S704_BT_CODE_2027.RBT5_STANDARD_WELD_DATA := W#16#0;
   S704_BT_CODE_2027.RBT6_STANDARD_WELD_DATA := W#16#0;
   S704_BT_CODE_2027.RBT7_STANDARD_WELD_DATA := W#16#0;
   S704_BT_CODE_2027.RBT8_STANDARD_WELD_DATA := W#16#0;
   S704_BT_CODE_2027.RBT9_STANDARD_WELD_DATA := W#16#0;
   S704_BT_CODE_2027.RBT10_STANDARD_WELD_DATA := W#16#0;
   S704_BT_CODE_2027.RBT11_STANDARD_WELD_DATA := W#16#0;
   S704_BT_CODE_2027.RBT12_STANDARD_WELD_DATA := W#16#0;
   S704_BT_CODE_2027.RBT13_STANDARD_WELD_DATA := W#16#0;
   S704_BT_CODE_2027.RBT14_STANDARD_WELD_DATA := W#16#0;
   S704_BT_CODE_2027.RBT15_STANDARD_WELD_DATA := W#16#0;
   S704_BT_CODE_2027.RBT16_STANDARD_WELD_DATA := W#16#0;
   S704_BT_CODE_2027.RBT17_STANDARD_WELD_DATA := W#16#0;
   S704_BT_CODE_2027.RBT18_STANDARD_WELD_DATA := W#16#0;
   S704_BT_CODE_2027.RBT19_STANDARD_WELD_DATA := W#16#0;
   S704_BT_CODE_2027.RBT20_STANDARD_WELD_DATA := W#16#0;
   S704_BT_CODE_2027.RBT21_STANDARD_WELD_DATA := W#16#0;
   S704_BT_CODE_2027.RBT22_STANDARD_WELD_DATA := W#16#0;
   S704_BT_CODE_2027.RBT23_STANDARD_WELD_DAT := W#16#0;
   S704_BT_CODE_2027.RBT24_STANDARD_WELD_DAT := W#16#0;
   S704_BT_CODE_2027.CHK_WORD := W#16#0;
   S704_BT_CODE_2027.TEST_TEMP[1] := B#16#0;
   S704_BT_CODE_2027.TEST_TEMP[2] := B#16#0;
   S704_BT_CODE_2027.TEST_TEMP[3] := B#16#0;
   S704_BT_CODE_2027.TEST_TEMP[4] := B#16#0;
   S704_BT_CODE_2027.TEST_TEMP[5] := B#16#0;
   S704_BT_CODE_2027.TEST_TEMP[6] := B#16#0;
   S704_BT_CODE_2027.TEST_TEMP[7] := B#16#0;
   S704_BT_CODE_2027.TEST_TEMP[8] := B#16#0;
   S704_BT_CODE_2027.TEST_TEMP[9] := B#16#0;
   S704_BT_CODE_2027.TEST_TEMP[10] := B#16#0;
   S704_BT_CODE_2027.TEST_TEMP[11] := B#16#0;
   S704_BT_CODE_2027.TEST_TEMP[12] := B#16#0;
   S704_BT_CODE_2027.TEST_TEMP[13] := B#16#0;
   S704_BT_CODE_2027.TEST_TEMP[14] := B#16#0;
   S704_BT_CODE_2027.TEST_TEMP[15] := B#16#0;
   S704_BT_CODE_2027.TEST_TEMP[16] := B#16#0;
   S704_BT_CODE_2027.TEST_TEMP[17] := B#16#0;
   S704_BT_CODE_2027.TEST_TEMP[18] := B#16#0;
   S704_BT_CODE_2027.TEST_TEMP[19] := B#16#0;
   S704_BT_CODE_2027.TEST_TEMP[20] := B#16#0;
   S704_BT_CODE_2027.TEST_TEMP[21] := B#16#0;
   S704_BT_CODE_2027.TEST_TEMP[22] := B#16#0;
   S704_BT_CODE_2027.TEST_TEMP[23] := B#16#0;
   S704_BT_CODE_2027.TEST_TEMP[24] := B#16#0;
   S704_BT_CODE_2027.TEST_TEMP[25] := B#16#0;
   S704_BT_CODE_2027.TEST_TEMP[26] := B#16#0;
   S704_BT_CODE_2027.TEST_TEMP[27] := B#16#0;
   S704_BT_CODE_2027.TEST_TEMP[28] := B#16#0;
   S704_BT_CODE_2027.TEST_TEMP[29] := B#16#0;
   S704_BT_CODE_2027.TEST_TEMP[30] := B#16#0;
   S704_BT_CODE_2027.TEST_TEMP[31] := B#16#0;
   S704_BT_CODE_2027.TEST_TEMP[32] := B#16#0;
   S704_BT_CODE_2027.TEST_TEMP[33] := B#16#0;
   S704_BT_CODE_2027.TEST_TEMP[34] := B#16#0;
   S704_BT_CODE_2027.TEST_TEMP[35] := B#16#0;
   S704_BT_CODE_2027.TEST_TEMP[36] := B#16#0;
   S704_BT_CODE_2027.TEST_TEMP[37] := B#16#0;
   S704_BT_CODE_2027.TEST_TEMP[38] := B#16#0;
   S704_BT_CODE_2027.TEST_TEMP[39] := B#16#0;
   S704_BT_CODE_2027.TEST_TEMP[40] := B#16#0;
   S704_BT_CODE_2028.STATION_MAIN := W#16#0;
   S704_BT_CODE_2028.DISTINCTION_LH_RH := W#16#0;
   S704_BT_CODE_2028.STAION_NUMBER := W#16#0;
   S704_BT_CODE_2028.BODY_TYPE_1ST := W#16#0;
   S704_BT_CODE_2028.BODY_TYPE_OPTION := W#16#0;
   S704_BT_CODE_2028.RBT1_STANDARD_WELD_DATA := W#16#0;
   S704_BT_CODE_2028.RBT2_STANDARD_WELD_DATA := W#16#0;
   S704_BT_CODE_2028.RBT3_STANDARD_WELD_DATA := W#16#0;
   S704_BT_CODE_2028.RBT4_STANDARD_WELD_DATA := W#16#0;
   S704_BT_CODE_2028.RBT5_STANDARD_WELD_DATA := W#16#0;
   S704_BT_CODE_2028.RBT6_STANDARD_WELD_DATA := W#16#0;
   S704_BT_CODE_2028.RBT7_STANDARD_WELD_DATA := W#16#0;
   S704_BT_CODE_2028.RBT8_STANDARD_WELD_DATA := W#16#0;
   S704_BT_CODE_2028.RBT9_STANDARD_WELD_DATA := W#16#0;
   S704_BT_CODE_2028.RBT10_STANDARD_WELD_DATA := W#16#0;
   S704_BT_CODE_2028.RBT11_STANDARD_WELD_DATA := W#16#0;
   S704_BT_CODE_2028.RBT12_STANDARD_WELD_DATA := W#16#0;
   S704_BT_CODE_2028.RBT13_STANDARD_WELD_DATA := W#16#0;
   S704_BT_CODE_2028.RBT14_STANDARD_WELD_DATA := W#16#0;
   S704_BT_CODE_2028.RBT15_STANDARD_WELD_DATA := W#16#0;
   S704_BT_CODE_2028.RBT16_STANDARD_WELD_DATA := W#16#0;
   S704_BT_CODE_2028.RBT17_STANDARD_WELD_DATA := W#16#0;
   S704_BT_CODE_2028.RBT18_STANDARD_WELD_DATA := W#16#0;
   S704_BT_CODE_2028.RBT19_STANDARD_WELD_DATA := W#16#0;
   S704_BT_CODE_2028.RBT20_STANDARD_WELD_DATA := W#16#0;
   S704_BT_CODE_2028.RBT21_STANDARD_WELD_DATA := W#16#0;
   S704_BT_CODE_2028.RBT22_STANDARD_WELD_DATA := W#16#0;
   S704_BT_CODE_2028.RBT23_STANDARD_WELD_DAT := W#16#0;
   S704_BT_CODE_2028.RBT24_STANDARD_WELD_DAT := W#16#0;
   S704_BT_CODE_2028.CHK_WORD := W#16#0;
   S704_BT_CODE_2028.TEST_TEMP[1] := B#16#0;
   S704_BT_CODE_2028.TEST_TEMP[2] := B#16#0;
   S704_BT_CODE_2028.TEST_TEMP[3] := B#16#0;
   S704_BT_CODE_2028.TEST_TEMP[4] := B#16#0;
   S704_BT_CODE_2028.TEST_TEMP[5] := B#16#0;
   S704_BT_CODE_2028.TEST_TEMP[6] := B#16#0;
   S704_BT_CODE_2028.TEST_TEMP[7] := B#16#0;
   S704_BT_CODE_2028.TEST_TEMP[8] := B#16#0;
   S704_BT_CODE_2028.TEST_TEMP[9] := B#16#0;
   S704_BT_CODE_2028.TEST_TEMP[10] := B#16#0;
   S704_BT_CODE_2028.TEST_TEMP[11] := B#16#0;
   S704_BT_CODE_2028.TEST_TEMP[12] := B#16#0;
   S704_BT_CODE_2028.TEST_TEMP[13] := B#16#0;
   S704_BT_CODE_2028.TEST_TEMP[14] := B#16#0;
   S704_BT_CODE_2028.TEST_TEMP[15] := B#16#0;
   S704_BT_CODE_2028.TEST_TEMP[16] := B#16#0;
   S704_BT_CODE_2028.TEST_TEMP[17] := B#16#0;
   S704_BT_CODE_2028.TEST_TEMP[18] := B#16#0;
   S704_BT_CODE_2028.TEST_TEMP[19] := B#16#0;
   S704_BT_CODE_2028.TEST_TEMP[20] := B#16#0;
   S704_BT_CODE_2028.TEST_TEMP[21] := B#16#0;
   S704_BT_CODE_2028.TEST_TEMP[22] := B#16#0;
   S704_BT_CODE_2028.TEST_TEMP[23] := B#16#0;
   S704_BT_CODE_2028.TEST_TEMP[24] := B#16#0;
   S704_BT_CODE_2028.TEST_TEMP[25] := B#16#0;
   S704_BT_CODE_2028.TEST_TEMP[26] := B#16#0;
   S704_BT_CODE_2028.TEST_TEMP[27] := B#16#0;
   S704_BT_CODE_2028.TEST_TEMP[28] := B#16#0;
   S704_BT_CODE_2028.TEST_TEMP[29] := B#16#0;
   S704_BT_CODE_2028.TEST_TEMP[30] := B#16#0;
   S704_BT_CODE_2028.TEST_TEMP[31] := B#16#0;
   S704_BT_CODE_2028.TEST_TEMP[32] := B#16#0;
   S704_BT_CODE_2028.TEST_TEMP[33] := B#16#0;
   S704_BT_CODE_2028.TEST_TEMP[34] := B#16#0;
   S704_BT_CODE_2028.TEST_TEMP[35] := B#16#0;
   S704_BT_CODE_2028.TEST_TEMP[36] := B#16#0;
   S704_BT_CODE_2028.TEST_TEMP[37] := B#16#0;
   S704_BT_CODE_2028.TEST_TEMP[38] := B#16#0;
   S704_BT_CODE_2028.TEST_TEMP[39] := B#16#0;
   S704_BT_CODE_2028.TEST_TEMP[40] := B#16#0;
   S704_BT_CODE_2029.STATION_MAIN := W#16#0;
   S704_BT_CODE_2029.DISTINCTION_LH_RH := W#16#0;
   S704_BT_CODE_2029.STAION_NUMBER := W#16#0;
   S704_BT_CODE_2029.BODY_TYPE_1ST := W#16#0;
   S704_BT_CODE_2029.BODY_TYPE_OPTION := W#16#0;
   S704_BT_CODE_2029.RBT1_STANDARD_WELD_DATA := W#16#0;
   S704_BT_CODE_2029.RBT2_STANDARD_WELD_DATA := W#16#0;
   S704_BT_CODE_2029.RBT3_STANDARD_WELD_DATA := W#16#0;
   S704_BT_CODE_2029.RBT4_STANDARD_WELD_DATA := W#16#0;
   S704_BT_CODE_2029.RBT5_STANDARD_WELD_DATA := W#16#0;
   S704_BT_CODE_2029.RBT6_STANDARD_WELD_DATA := W#16#0;
   S704_BT_CODE_2029.RBT7_STANDARD_WELD_DATA := W#16#0;
   S704_BT_CODE_2029.RBT8_STANDARD_WELD_DATA := W#16#0;
   S704_BT_CODE_2029.RBT9_STANDARD_WELD_DATA := W#16#0;
   S704_BT_CODE_2029.RBT10_STANDARD_WELD_DATA := W#16#0;
   S704_BT_CODE_2029.RBT11_STANDARD_WELD_DATA := W#16#0;
   S704_BT_CODE_2029.RBT12_STANDARD_WELD_DATA := W#16#0;
   S704_BT_CODE_2029.RBT13_STANDARD_WELD_DATA := W#16#0;
   S704_BT_CODE_2029.RBT14_STANDARD_WELD_DATA := W#16#0;
   S704_BT_CODE_2029.RBT15_STANDARD_WELD_DATA := W#16#0;
   S704_BT_CODE_2029.RBT16_STANDARD_WELD_DATA := W#16#0;
   S704_BT_CODE_2029.RBT17_STANDARD_WELD_DATA := W#16#0;
   S704_BT_CODE_2029.RBT18_STANDARD_WELD_DATA := W#16#0;
   S704_BT_CODE_2029.RBT19_STANDARD_WELD_DATA := W#16#0;
   S704_BT_CODE_2029.RBT20_STANDARD_WELD_DATA := W#16#0;
   S704_BT_CODE_2029.RBT21_STANDARD_WELD_DATA := W#16#0;
   S704_BT_CODE_2029.RBT22_STANDARD_WELD_DATA := W#16#0;
   S704_BT_CODE_2029.RBT23_STANDARD_WELD_DAT := W#16#0;
   S704_BT_CODE_2029.RBT24_STANDARD_WELD_DAT := W#16#0;
   S704_BT_CODE_2029.CHK_WORD := W#16#0;
   S704_BT_CODE_2029.TEST_TEMP[1] := B#16#0;
   S704_BT_CODE_2029.TEST_TEMP[2] := B#16#0;
   S704_BT_CODE_2029.TEST_TEMP[3] := B#16#0;
   S704_BT_CODE_2029.TEST_TEMP[4] := B#16#0;
   S704_BT_CODE_2029.TEST_TEMP[5] := B#16#0;
   S704_BT_CODE_2029.TEST_TEMP[6] := B#16#0;
   S704_BT_CODE_2029.TEST_TEMP[7] := B#16#0;
   S704_BT_CODE_2029.TEST_TEMP[8] := B#16#0;
   S704_BT_CODE_2029.TEST_TEMP[9] := B#16#0;
   S704_BT_CODE_2029.TEST_TEMP[10] := B#16#0;
   S704_BT_CODE_2029.TEST_TEMP[11] := B#16#0;
   S704_BT_CODE_2029.TEST_TEMP[12] := B#16#0;
   S704_BT_CODE_2029.TEST_TEMP[13] := B#16#0;
   S704_BT_CODE_2029.TEST_TEMP[14] := B#16#0;
   S704_BT_CODE_2029.TEST_TEMP[15] := B#16#0;
   S704_BT_CODE_2029.TEST_TEMP[16] := B#16#0;
   S704_BT_CODE_2029.TEST_TEMP[17] := B#16#0;
   S704_BT_CODE_2029.TEST_TEMP[18] := B#16#0;
   S704_BT_CODE_2029.TEST_TEMP[19] := B#16#0;
   S704_BT_CODE_2029.TEST_TEMP[20] := B#16#0;
   S704_BT_CODE_2029.TEST_TEMP[21] := B#16#0;
   S704_BT_CODE_2029.TEST_TEMP[22] := B#16#0;
   S704_BT_CODE_2029.TEST_TEMP[23] := B#16#0;
   S704_BT_CODE_2029.TEST_TEMP[24] := B#16#0;
   S704_BT_CODE_2029.TEST_TEMP[25] := B#16#0;
   S704_BT_CODE_2029.TEST_TEMP[26] := B#16#0;
   S704_BT_CODE_2029.TEST_TEMP[27] := B#16#0;
   S704_BT_CODE_2029.TEST_TEMP[28] := B#16#0;
   S704_BT_CODE_2029.TEST_TEMP[29] := B#16#0;
   S704_BT_CODE_2029.TEST_TEMP[30] := B#16#0;
   S704_BT_CODE_2029.TEST_TEMP[31] := B#16#0;
   S704_BT_CODE_2029.TEST_TEMP[32] := B#16#0;
   S704_BT_CODE_2029.TEST_TEMP[33] := B#16#0;
   S704_BT_CODE_2029.TEST_TEMP[34] := B#16#0;
   S704_BT_CODE_2029.TEST_TEMP[35] := B#16#0;
   S704_BT_CODE_2029.TEST_TEMP[36] := B#16#0;
   S704_BT_CODE_2029.TEST_TEMP[37] := B#16#0;
   S704_BT_CODE_2029.TEST_TEMP[38] := B#16#0;
   S704_BT_CODE_2029.TEST_TEMP[39] := B#16#0;
   S704_BT_CODE_2029.TEST_TEMP[40] := B#16#0;
   S704_BT_CODE_2030.STATION_MAIN := W#16#0;
   S704_BT_CODE_2030.DISTINCTION_LH_RH := W#16#0;
   S704_BT_CODE_2030.STAION_NUMBER := W#16#0;
   S704_BT_CODE_2030.BODY_TYPE_1ST := W#16#0;
   S704_BT_CODE_2030.BODY_TYPE_OPTION := W#16#0;
   S704_BT_CODE_2030.RBT1_STANDARD_WELD_DATA := W#16#0;
   S704_BT_CODE_2030.RBT2_STANDARD_WELD_DATA := W#16#0;
   S704_BT_CODE_2030.RBT3_STANDARD_WELD_DATA := W#16#0;
   S704_BT_CODE_2030.RBT4_STANDARD_WELD_DATA := W#16#0;
   S704_BT_CODE_2030.RBT5_STANDARD_WELD_DATA := W#16#0;
   S704_BT_CODE_2030.RBT6_STANDARD_WELD_DATA := W#16#0;
   S704_BT_CODE_2030.RBT7_STANDARD_WELD_DATA := W#16#0;
   S704_BT_CODE_2030.RBT8_STANDARD_WELD_DATA := W#16#0;
   S704_BT_CODE_2030.RBT9_STANDARD_WELD_DATA := W#16#0;
   S704_BT_CODE_2030.RBT10_STANDARD_WELD_DATA := W#16#0;
   S704_BT_CODE_2030.RBT11_STANDARD_WELD_DATA := W#16#0;
   S704_BT_CODE_2030.RBT12_STANDARD_WELD_DATA := W#16#0;
   S704_BT_CODE_2030.RBT13_STANDARD_WELD_DATA := W#16#0;
   S704_BT_CODE_2030.RBT14_STANDARD_WELD_DATA := W#16#0;
   S704_BT_CODE_2030.RBT15_STANDARD_WELD_DATA := W#16#0;
   S704_BT_CODE_2030.RBT16_STANDARD_WELD_DATA := W#16#0;
   S704_BT_CODE_2030.RBT17_STANDARD_WELD_DATA := W#16#0;
   S704_BT_CODE_2030.RBT18_STANDARD_WELD_DATA := W#16#0;
   S704_BT_CODE_2030.RBT19_STANDARD_WELD_DATA := W#16#0;
   S704_BT_CODE_2030.RBT20_STANDARD_WELD_DATA := W#16#0;
   S704_BT_CODE_2030.RBT21_STANDARD_WELD_DATA := W#16#0;
   S704_BT_CODE_2030.RBT22_STANDARD_WELD_DATA := W#16#0;
   S704_BT_CODE_2030.RBT23_STANDARD_WELD_DAT := W#16#0;
   S704_BT_CODE_2030.RBT24_STANDARD_WELD_DAT := W#16#0;
   S704_BT_CODE_2030.CHK_WORD := W#16#0;
   S704_BT_CODE_2030.TEST_TEMP[1] := B#16#0;
   S704_BT_CODE_2030.TEST_TEMP[2] := B#16#0;
   S704_BT_CODE_2030.TEST_TEMP[3] := B#16#0;
   S704_BT_CODE_2030.TEST_TEMP[4] := B#16#0;
   S704_BT_CODE_2030.TEST_TEMP[5] := B#16#0;
   S704_BT_CODE_2030.TEST_TEMP[6] := B#16#0;
   S704_BT_CODE_2030.TEST_TEMP[7] := B#16#0;
   S704_BT_CODE_2030.TEST_TEMP[8] := B#16#0;
   S704_BT_CODE_2030.TEST_TEMP[9] := B#16#0;
   S704_BT_CODE_2030.TEST_TEMP[10] := B#16#0;
   S704_BT_CODE_2030.TEST_TEMP[11] := B#16#0;
   S704_BT_CODE_2030.TEST_TEMP[12] := B#16#0;
   S704_BT_CODE_2030.TEST_TEMP[13] := B#16#0;
   S704_BT_CODE_2030.TEST_TEMP[14] := B#16#0;
   S704_BT_CODE_2030.TEST_TEMP[15] := B#16#0;
   S704_BT_CODE_2030.TEST_TEMP[16] := B#16#0;
   S704_BT_CODE_2030.TEST_TEMP[17] := B#16#0;
   S704_BT_CODE_2030.TEST_TEMP[18] := B#16#0;
   S704_BT_CODE_2030.TEST_TEMP[19] := B#16#0;
   S704_BT_CODE_2030.TEST_TEMP[20] := B#16#0;
   S704_BT_CODE_2030.TEST_TEMP[21] := B#16#0;
   S704_BT_CODE_2030.TEST_TEMP[22] := B#16#0;
   S704_BT_CODE_2030.TEST_TEMP[23] := B#16#0;
   S704_BT_CODE_2030.TEST_TEMP[24] := B#16#0;
   S704_BT_CODE_2030.TEST_TEMP[25] := B#16#0;
   S704_BT_CODE_2030.TEST_TEMP[26] := B#16#0;
   S704_BT_CODE_2030.TEST_TEMP[27] := B#16#0;
   S704_BT_CODE_2030.TEST_TEMP[28] := B#16#0;
   S704_BT_CODE_2030.TEST_TEMP[29] := B#16#0;
   S704_BT_CODE_2030.TEST_TEMP[30] := B#16#0;
   S704_BT_CODE_2030.TEST_TEMP[31] := B#16#0;
   S704_BT_CODE_2030.TEST_TEMP[32] := B#16#0;
   S704_BT_CODE_2030.TEST_TEMP[33] := B#16#0;
   S704_BT_CODE_2030.TEST_TEMP[34] := B#16#0;
   S704_BT_CODE_2030.TEST_TEMP[35] := B#16#0;
   S704_BT_CODE_2030.TEST_TEMP[36] := B#16#0;
   S704_BT_CODE_2030.TEST_TEMP[37] := B#16#0;
   S704_BT_CODE_2030.TEST_TEMP[38] := B#16#0;
   S704_BT_CODE_2030.TEST_TEMP[39] := B#16#0;
   S704_BT_CODE_2030.TEST_TEMP[40] := B#16#0;
   S702_BT_CODE_2101.STATION_MAIN := W#16#0;
   S702_BT_CODE_2101.DISTINCTION_LH_RH := W#16#0;
   S702_BT_CODE_2101.STAION_NUMBER := W#16#0;
   S702_BT_CODE_2101.BODY_TYPE_1ST := W#16#0;
   S702_BT_CODE_2101.BODY_TYPE_OPTION := W#16#0;
   S702_BT_CODE_2101.RBT1_STANDARD_WELD_DATA := W#16#0;
   S702_BT_CODE_2101.RBT2_STANDARD_WELD_DATA := W#16#0;
   S702_BT_CODE_2101.RBT3_STANDARD_WELD_DATA := W#16#0;
   S702_BT_CODE_2101.RBT4_STANDARD_WELD_DATA := W#16#0;
   S702_BT_CODE_2101.RBT5_STANDARD_WELD_DATA := W#16#0;
   S702_BT_CODE_2101.RBT6_STANDARD_WELD_DATA := W#16#0;
   S702_BT_CODE_2101.RBT7_STANDARD_WELD_DATA := W#16#0;
   S702_BT_CODE_2101.RBT8_STANDARD_WELD_DATA := W#16#0;
   S702_BT_CODE_2101.RBT9_STANDARD_WELD_DATA := W#16#0;
   S702_BT_CODE_2101.RBT10_STANDARD_WELD_DATA := W#16#0;
   S702_BT_CODE_2101.RBT11_STANDARD_WELD_DATA := W#16#0;
   S702_BT_CODE_2101.RBT12_STANDARD_WELD_DATA := W#16#0;
   S702_BT_CODE_2101.RBT13_STANDARD_WELD_DATA := W#16#0;
   S702_BT_CODE_2101.RBT14_STANDARD_WELD_DATA := W#16#0;
   S702_BT_CODE_2101.RBT15_STANDARD_WELD_DATA := W#16#0;
   S702_BT_CODE_2101.RBT16_STANDARD_WELD_DATA := W#16#0;
   S702_BT_CODE_2101.RBT17_STANDARD_WELD_DATA := W#16#0;
   S702_BT_CODE_2101.RBT18_STANDARD_WELD_DATA := W#16#0;
   S702_BT_CODE_2101.RBT19_STANDARD_WELD_DATA := W#16#0;
   S702_BT_CODE_2101.RBT20_STANDARD_WELD_DATA := W#16#0;
   S702_BT_CODE_2101.RBT21_STANDARD_WELD_DATA := W#16#0;
   S702_BT_CODE_2101.RBT22_STANDARD_WELD_DATA := W#16#0;
   S702_BT_CODE_2101.RBT23_STANDARD_WELD_DAT := W#16#0;
   S702_BT_CODE_2101.RBT24_STANDARD_WELD_DAT := W#16#0;
   S702_BT_CODE_2101.CHK_WORD := W#16#0;
   S702_BT_CODE_2101.TEST_TEMP[1] := B#16#0;
   S702_BT_CODE_2101.TEST_TEMP[2] := B#16#0;
   S702_BT_CODE_2101.TEST_TEMP[3] := B#16#0;
   S702_BT_CODE_2101.TEST_TEMP[4] := B#16#0;
   S702_BT_CODE_2101.TEST_TEMP[5] := B#16#0;
   S702_BT_CODE_2101.TEST_TEMP[6] := B#16#0;
   S702_BT_CODE_2101.TEST_TEMP[7] := B#16#0;
   S702_BT_CODE_2101.TEST_TEMP[8] := B#16#0;
   S702_BT_CODE_2101.TEST_TEMP[9] := B#16#0;
   S702_BT_CODE_2101.TEST_TEMP[10] := B#16#0;
   S702_BT_CODE_2101.TEST_TEMP[11] := B#16#0;
   S702_BT_CODE_2101.TEST_TEMP[12] := B#16#0;
   S702_BT_CODE_2101.TEST_TEMP[13] := B#16#0;
   S702_BT_CODE_2101.TEST_TEMP[14] := B#16#0;
   S702_BT_CODE_2101.TEST_TEMP[15] := B#16#0;
   S702_BT_CODE_2101.TEST_TEMP[16] := B#16#0;
   S702_BT_CODE_2101.TEST_TEMP[17] := B#16#0;
   S702_BT_CODE_2101.TEST_TEMP[18] := B#16#0;
   S702_BT_CODE_2101.TEST_TEMP[19] := B#16#0;
   S702_BT_CODE_2101.TEST_TEMP[20] := B#16#0;
   S702_BT_CODE_2101.TEST_TEMP[21] := B#16#0;
   S702_BT_CODE_2101.TEST_TEMP[22] := B#16#0;
   S702_BT_CODE_2101.TEST_TEMP[23] := B#16#0;
   S702_BT_CODE_2101.TEST_TEMP[24] := B#16#0;
   S702_BT_CODE_2101.TEST_TEMP[25] := B#16#0;
   S702_BT_CODE_2101.TEST_TEMP[26] := B#16#0;
   S702_BT_CODE_2101.TEST_TEMP[27] := B#16#0;
   S702_BT_CODE_2101.TEST_TEMP[28] := B#16#0;
   S702_BT_CODE_2101.TEST_TEMP[29] := B#16#0;
   S702_BT_CODE_2101.TEST_TEMP[30] := B#16#0;
   S702_BT_CODE_2101.TEST_TEMP[31] := B#16#0;
   S702_BT_CODE_2101.TEST_TEMP[32] := B#16#0;
   S702_BT_CODE_2101.TEST_TEMP[33] := B#16#0;
   S702_BT_CODE_2101.TEST_TEMP[34] := B#16#0;
   S702_BT_CODE_2101.TEST_TEMP[35] := B#16#0;
   S702_BT_CODE_2101.TEST_TEMP[36] := B#16#0;
   S702_BT_CODE_2101.TEST_TEMP[37] := B#16#0;
   S702_BT_CODE_2101.TEST_TEMP[38] := B#16#0;
   S702_BT_CODE_2101.TEST_TEMP[39] := B#16#0;
   S702_BT_CODE_2101.TEST_TEMP[40] := B#16#0;
   S702_BT_CODE_2102.STATION_MAIN := W#16#0;
   S702_BT_CODE_2102.DISTINCTION_LH_RH := W#16#0;
   S702_BT_CODE_2102.STAION_NUMBER := W#16#0;
   S702_BT_CODE_2102.BODY_TYPE_1ST := W#16#0;
   S702_BT_CODE_2102.BODY_TYPE_OPTION := W#16#0;
   S702_BT_CODE_2102.RBT1_STANDARD_WELD_DATA := W#16#0;
   S702_BT_CODE_2102.RBT2_STANDARD_WELD_DATA := W#16#0;
   S702_BT_CODE_2102.RBT3_STANDARD_WELD_DATA := W#16#0;
   S702_BT_CODE_2102.RBT4_STANDARD_WELD_DATA := W#16#0;
   S702_BT_CODE_2102.RBT5_STANDARD_WELD_DATA := W#16#0;
   S702_BT_CODE_2102.RBT6_STANDARD_WELD_DATA := W#16#0;
   S702_BT_CODE_2102.RBT7_STANDARD_WELD_DATA := W#16#0;
   S702_BT_CODE_2102.RBT8_STANDARD_WELD_DATA := W#16#0;
   S702_BT_CODE_2102.RBT9_STANDARD_WELD_DATA := W#16#0;
   S702_BT_CODE_2102.RBT10_STANDARD_WELD_DATA := W#16#0;
   S702_BT_CODE_2102.RBT11_STANDARD_WELD_DATA := W#16#0;
   S702_BT_CODE_2102.RBT12_STANDARD_WELD_DATA := W#16#0;
   S702_BT_CODE_2102.RBT13_STANDARD_WELD_DATA := W#16#0;
   S702_BT_CODE_2102.RBT14_STANDARD_WELD_DATA := W#16#0;
   S702_BT_CODE_2102.RBT15_STANDARD_WELD_DATA := W#16#0;
   S702_BT_CODE_2102.RBT16_STANDARD_WELD_DATA := W#16#0;
   S702_BT_CODE_2102.RBT17_STANDARD_WELD_DATA := W#16#0;
   S702_BT_CODE_2102.RBT18_STANDARD_WELD_DATA := W#16#0;
   S702_BT_CODE_2102.RBT19_STANDARD_WELD_DATA := W#16#0;
   S702_BT_CODE_2102.RBT20_STANDARD_WELD_DATA := W#16#0;
   S702_BT_CODE_2102.RBT21_STANDARD_WELD_DATA := W#16#0;
   S702_BT_CODE_2102.RBT22_STANDARD_WELD_DATA := W#16#0;
   S702_BT_CODE_2102.RBT23_STANDARD_WELD_DAT := W#16#0;
   S702_BT_CODE_2102.RBT24_STANDARD_WELD_DAT := W#16#0;
   S702_BT_CODE_2102.CHK_WORD := W#16#0;
   S702_BT_CODE_2102.TEST_TEMP[1] := B#16#0;
   S702_BT_CODE_2102.TEST_TEMP[2] := B#16#0;
   S702_BT_CODE_2102.TEST_TEMP[3] := B#16#0;
   S702_BT_CODE_2102.TEST_TEMP[4] := B#16#0;
   S702_BT_CODE_2102.TEST_TEMP[5] := B#16#0;
   S702_BT_CODE_2102.TEST_TEMP[6] := B#16#0;
   S702_BT_CODE_2102.TEST_TEMP[7] := B#16#0;
   S702_BT_CODE_2102.TEST_TEMP[8] := B#16#0;
   S702_BT_CODE_2102.TEST_TEMP[9] := B#16#0;
   S702_BT_CODE_2102.TEST_TEMP[10] := B#16#0;
   S702_BT_CODE_2102.TEST_TEMP[11] := B#16#0;
   S702_BT_CODE_2102.TEST_TEMP[12] := B#16#0;
   S702_BT_CODE_2102.TEST_TEMP[13] := B#16#0;
   S702_BT_CODE_2102.TEST_TEMP[14] := B#16#0;
   S702_BT_CODE_2102.TEST_TEMP[15] := B#16#0;
   S702_BT_CODE_2102.TEST_TEMP[16] := B#16#0;
   S702_BT_CODE_2102.TEST_TEMP[17] := B#16#0;
   S702_BT_CODE_2102.TEST_TEMP[18] := B#16#0;
   S702_BT_CODE_2102.TEST_TEMP[19] := B#16#0;
   S702_BT_CODE_2102.TEST_TEMP[20] := B#16#0;
   S702_BT_CODE_2102.TEST_TEMP[21] := B#16#0;
   S702_BT_CODE_2102.TEST_TEMP[22] := B#16#0;
   S702_BT_CODE_2102.TEST_TEMP[23] := B#16#0;
   S702_BT_CODE_2102.TEST_TEMP[24] := B#16#0;
   S702_BT_CODE_2102.TEST_TEMP[25] := B#16#0;
   S702_BT_CODE_2102.TEST_TEMP[26] := B#16#0;
   S702_BT_CODE_2102.TEST_TEMP[27] := B#16#0;
   S702_BT_CODE_2102.TEST_TEMP[28] := B#16#0;
   S702_BT_CODE_2102.TEST_TEMP[29] := B#16#0;
   S702_BT_CODE_2102.TEST_TEMP[30] := B#16#0;
   S702_BT_CODE_2102.TEST_TEMP[31] := B#16#0;
   S702_BT_CODE_2102.TEST_TEMP[32] := B#16#0;
   S702_BT_CODE_2102.TEST_TEMP[33] := B#16#0;
   S702_BT_CODE_2102.TEST_TEMP[34] := B#16#0;
   S702_BT_CODE_2102.TEST_TEMP[35] := B#16#0;
   S702_BT_CODE_2102.TEST_TEMP[36] := B#16#0;
   S702_BT_CODE_2102.TEST_TEMP[37] := B#16#0;
   S702_BT_CODE_2102.TEST_TEMP[38] := B#16#0;
   S702_BT_CODE_2102.TEST_TEMP[39] := B#16#0;
   S702_BT_CODE_2102.TEST_TEMP[40] := B#16#0;
   S702_BT_CODE_2103.STATION_MAIN := W#16#0;
   S702_BT_CODE_2103.DISTINCTION_LH_RH := W#16#0;
   S702_BT_CODE_2103.STAION_NUMBER := W#16#0;
   S702_BT_CODE_2103.BODY_TYPE_1ST := W#16#0;
   S702_BT_CODE_2103.BODY_TYPE_OPTION := W#16#0;
   S702_BT_CODE_2103.RBT1_STANDARD_WELD_DATA := W#16#0;
   S702_BT_CODE_2103.RBT2_STANDARD_WELD_DATA := W#16#0;
   S702_BT_CODE_2103.RBT3_STANDARD_WELD_DATA := W#16#0;
   S702_BT_CODE_2103.RBT4_STANDARD_WELD_DATA := W#16#0;
   S702_BT_CODE_2103.RBT5_STANDARD_WELD_DATA := W#16#0;
   S702_BT_CODE_2103.RBT6_STANDARD_WELD_DATA := W#16#0;
   S702_BT_CODE_2103.RBT7_STANDARD_WELD_DATA := W#16#0;
   S702_BT_CODE_2103.RBT8_STANDARD_WELD_DATA := W#16#0;
   S702_BT_CODE_2103.RBT9_STANDARD_WELD_DATA := W#16#0;
   S702_BT_CODE_2103.RBT10_STANDARD_WELD_DATA := W#16#0;
   S702_BT_CODE_2103.RBT11_STANDARD_WELD_DATA := W#16#0;
   S702_BT_CODE_2103.RBT12_STANDARD_WELD_DATA := W#16#0;
   S702_BT_CODE_2103.RBT13_STANDARD_WELD_DATA := W#16#0;
   S702_BT_CODE_2103.RBT14_STANDARD_WELD_DATA := W#16#0;
   S702_BT_CODE_2103.RBT15_STANDARD_WELD_DATA := W#16#0;
   S702_BT_CODE_2103.RBT16_STANDARD_WELD_DATA := W#16#0;
   S702_BT_CODE_2103.RBT17_STANDARD_WELD_DATA := W#16#0;
   S702_BT_CODE_2103.RBT18_STANDARD_WELD_DATA := W#16#0;
   S702_BT_CODE_2103.RBT19_STANDARD_WELD_DATA := W#16#0;
   S702_BT_CODE_2103.RBT20_STANDARD_WELD_DATA := W#16#0;
   S702_BT_CODE_2103.RBT21_STANDARD_WELD_DATA := W#16#0;
   S702_BT_CODE_2103.RBT22_STANDARD_WELD_DATA := W#16#0;
   S702_BT_CODE_2103.RBT23_STANDARD_WELD_DAT := W#16#0;
   S702_BT_CODE_2103.RBT24_STANDARD_WELD_DAT := W#16#0;
   S702_BT_CODE_2103.CHK_WORD := W#16#0;
   S702_BT_CODE_2103.TEST_TEMP[1] := B#16#0;
   S702_BT_CODE_2103.TEST_TEMP[2] := B#16#0;
   S702_BT_CODE_2103.TEST_TEMP[3] := B#16#0;
   S702_BT_CODE_2103.TEST_TEMP[4] := B#16#0;
   S702_BT_CODE_2103.TEST_TEMP[5] := B#16#0;
   S702_BT_CODE_2103.TEST_TEMP[6] := B#16#0;
   S702_BT_CODE_2103.TEST_TEMP[7] := B#16#0;
   S702_BT_CODE_2103.TEST_TEMP[8] := B#16#0;
   S702_BT_CODE_2103.TEST_TEMP[9] := B#16#0;
   S702_BT_CODE_2103.TEST_TEMP[10] := B#16#0;
   S702_BT_CODE_2103.TEST_TEMP[11] := B#16#0;
   S702_BT_CODE_2103.TEST_TEMP[12] := B#16#0;
   S702_BT_CODE_2103.TEST_TEMP[13] := B#16#0;
   S702_BT_CODE_2103.TEST_TEMP[14] := B#16#0;
   S702_BT_CODE_2103.TEST_TEMP[15] := B#16#0;
   S702_BT_CODE_2103.TEST_TEMP[16] := B#16#0;
   S702_BT_CODE_2103.TEST_TEMP[17] := B#16#0;
   S702_BT_CODE_2103.TEST_TEMP[18] := B#16#0;
   S702_BT_CODE_2103.TEST_TEMP[19] := B#16#0;
   S702_BT_CODE_2103.TEST_TEMP[20] := B#16#0;
   S702_BT_CODE_2103.TEST_TEMP[21] := B#16#0;
   S702_BT_CODE_2103.TEST_TEMP[22] := B#16#0;
   S702_BT_CODE_2103.TEST_TEMP[23] := B#16#0;
   S702_BT_CODE_2103.TEST_TEMP[24] := B#16#0;
   S702_BT_CODE_2103.TEST_TEMP[25] := B#16#0;
   S702_BT_CODE_2103.TEST_TEMP[26] := B#16#0;
   S702_BT_CODE_2103.TEST_TEMP[27] := B#16#0;
   S702_BT_CODE_2103.TEST_TEMP[28] := B#16#0;
   S702_BT_CODE_2103.TEST_TEMP[29] := B#16#0;
   S702_BT_CODE_2103.TEST_TEMP[30] := B#16#0;
   S702_BT_CODE_2103.TEST_TEMP[31] := B#16#0;
   S702_BT_CODE_2103.TEST_TEMP[32] := B#16#0;
   S702_BT_CODE_2103.TEST_TEMP[33] := B#16#0;
   S702_BT_CODE_2103.TEST_TEMP[34] := B#16#0;
   S702_BT_CODE_2103.TEST_TEMP[35] := B#16#0;
   S702_BT_CODE_2103.TEST_TEMP[36] := B#16#0;
   S702_BT_CODE_2103.TEST_TEMP[37] := B#16#0;
   S702_BT_CODE_2103.TEST_TEMP[38] := B#16#0;
   S702_BT_CODE_2103.TEST_TEMP[39] := B#16#0;
   S702_BT_CODE_2103.TEST_TEMP[40] := B#16#0;
   S702_BT_CODE_2104.STATION_MAIN := W#16#0;
   S702_BT_CODE_2104.DISTINCTION_LH_RH := W#16#0;
   S702_BT_CODE_2104.STAION_NUMBER := W#16#0;
   S702_BT_CODE_2104.BODY_TYPE_1ST := W#16#0;
   S702_BT_CODE_2104.BODY_TYPE_OPTION := W#16#0;
   S702_BT_CODE_2104.RBT1_STANDARD_WELD_DATA := W#16#0;
   S702_BT_CODE_2104.RBT2_STANDARD_WELD_DATA := W#16#0;
   S702_BT_CODE_2104.RBT3_STANDARD_WELD_DATA := W#16#0;
   S702_BT_CODE_2104.RBT4_STANDARD_WELD_DATA := W#16#0;
   S702_BT_CODE_2104.RBT5_STANDARD_WELD_DATA := W#16#0;
   S702_BT_CODE_2104.RBT6_STANDARD_WELD_DATA := W#16#0;
   S702_BT_CODE_2104.RBT7_STANDARD_WELD_DATA := W#16#0;
   S702_BT_CODE_2104.RBT8_STANDARD_WELD_DATA := W#16#0;
   S702_BT_CODE_2104.RBT9_STANDARD_WELD_DATA := W#16#0;
   S702_BT_CODE_2104.RBT10_STANDARD_WELD_DATA := W#16#0;
   S702_BT_CODE_2104.RBT11_STANDARD_WELD_DATA := W#16#0;
   S702_BT_CODE_2104.RBT12_STANDARD_WELD_DATA := W#16#0;
   S702_BT_CODE_2104.RBT13_STANDARD_WELD_DATA := W#16#0;
   S702_BT_CODE_2104.RBT14_STANDARD_WELD_DATA := W#16#0;
   S702_BT_CODE_2104.RBT15_STANDARD_WELD_DATA := W#16#0;
   S702_BT_CODE_2104.RBT16_STANDARD_WELD_DATA := W#16#0;
   S702_BT_CODE_2104.RBT17_STANDARD_WELD_DATA := W#16#0;
   S702_BT_CODE_2104.RBT18_STANDARD_WELD_DATA := W#16#0;
   S702_BT_CODE_2104.RBT19_STANDARD_WELD_DATA := W#16#0;
   S702_BT_CODE_2104.RBT20_STANDARD_WELD_DATA := W#16#0;
   S702_BT_CODE_2104.RBT21_STANDARD_WELD_DATA := W#16#0;
   S702_BT_CODE_2104.RBT22_STANDARD_WELD_DATA := W#16#0;
   S702_BT_CODE_2104.RBT23_STANDARD_WELD_DAT := W#16#0;
   S702_BT_CODE_2104.RBT24_STANDARD_WELD_DAT := W#16#0;
   S702_BT_CODE_2104.CHK_WORD := W#16#0;
   S702_BT_CODE_2104.TEST_TEMP[1] := B#16#0;
   S702_BT_CODE_2104.TEST_TEMP[2] := B#16#0;
   S702_BT_CODE_2104.TEST_TEMP[3] := B#16#0;
   S702_BT_CODE_2104.TEST_TEMP[4] := B#16#0;
   S702_BT_CODE_2104.TEST_TEMP[5] := B#16#0;
   S702_BT_CODE_2104.TEST_TEMP[6] := B#16#0;
   S702_BT_CODE_2104.TEST_TEMP[7] := B#16#0;
   S702_BT_CODE_2104.TEST_TEMP[8] := B#16#0;
   S702_BT_CODE_2104.TEST_TEMP[9] := B#16#0;
   S702_BT_CODE_2104.TEST_TEMP[10] := B#16#0;
   S702_BT_CODE_2104.TEST_TEMP[11] := B#16#0;
   S702_BT_CODE_2104.TEST_TEMP[12] := B#16#0;
   S702_BT_CODE_2104.TEST_TEMP[13] := B#16#0;
   S702_BT_CODE_2104.TEST_TEMP[14] := B#16#0;
   S702_BT_CODE_2104.TEST_TEMP[15] := B#16#0;
   S702_BT_CODE_2104.TEST_TEMP[16] := B#16#0;
   S702_BT_CODE_2104.TEST_TEMP[17] := B#16#0;
   S702_BT_CODE_2104.TEST_TEMP[18] := B#16#0;
   S702_BT_CODE_2104.TEST_TEMP[19] := B#16#0;
   S702_BT_CODE_2104.TEST_TEMP[20] := B#16#0;
   S702_BT_CODE_2104.TEST_TEMP[21] := B#16#0;
   S702_BT_CODE_2104.TEST_TEMP[22] := B#16#0;
   S702_BT_CODE_2104.TEST_TEMP[23] := B#16#0;
   S702_BT_CODE_2104.TEST_TEMP[24] := B#16#0;
   S702_BT_CODE_2104.TEST_TEMP[25] := B#16#0;
   S702_BT_CODE_2104.TEST_TEMP[26] := B#16#0;
   S702_BT_CODE_2104.TEST_TEMP[27] := B#16#0;
   S702_BT_CODE_2104.TEST_TEMP[28] := B#16#0;
   S702_BT_CODE_2104.TEST_TEMP[29] := B#16#0;
   S702_BT_CODE_2104.TEST_TEMP[30] := B#16#0;
   S702_BT_CODE_2104.TEST_TEMP[31] := B#16#0;
   S702_BT_CODE_2104.TEST_TEMP[32] := B#16#0;
   S702_BT_CODE_2104.TEST_TEMP[33] := B#16#0;
   S702_BT_CODE_2104.TEST_TEMP[34] := B#16#0;
   S702_BT_CODE_2104.TEST_TEMP[35] := B#16#0;
   S702_BT_CODE_2104.TEST_TEMP[36] := B#16#0;
   S702_BT_CODE_2104.TEST_TEMP[37] := B#16#0;
   S702_BT_CODE_2104.TEST_TEMP[38] := B#16#0;
   S702_BT_CODE_2104.TEST_TEMP[39] := B#16#0;
   S702_BT_CODE_2104.TEST_TEMP[40] := B#16#0;
   S702_BT_CODE_2105.STATION_MAIN := W#16#0;
   S702_BT_CODE_2105.DISTINCTION_LH_RH := W#16#0;
   S702_BT_CODE_2105.STAION_NUMBER := W#16#0;
   S702_BT_CODE_2105.BODY_TYPE_1ST := W#16#0;
   S702_BT_CODE_2105.BODY_TYPE_OPTION := W#16#0;
   S702_BT_CODE_2105.RBT1_STANDARD_WELD_DATA := W#16#0;
   S702_BT_CODE_2105.RBT2_STANDARD_WELD_DATA := W#16#0;
   S702_BT_CODE_2105.RBT3_STANDARD_WELD_DATA := W#16#0;
   S702_BT_CODE_2105.RBT4_STANDARD_WELD_DATA := W#16#0;
   S702_BT_CODE_2105.RBT5_STANDARD_WELD_DATA := W#16#0;
   S702_BT_CODE_2105.RBT6_STANDARD_WELD_DATA := W#16#0;
   S702_BT_CODE_2105.RBT7_STANDARD_WELD_DATA := W#16#0;
   S702_BT_CODE_2105.RBT8_STANDARD_WELD_DATA := W#16#0;
   S702_BT_CODE_2105.RBT9_STANDARD_WELD_DATA := W#16#0;
   S702_BT_CODE_2105.RBT10_STANDARD_WELD_DATA := W#16#0;
   S702_BT_CODE_2105.RBT11_STANDARD_WELD_DATA := W#16#0;
   S702_BT_CODE_2105.RBT12_STANDARD_WELD_DATA := W#16#0;
   S702_BT_CODE_2105.RBT13_STANDARD_WELD_DATA := W#16#0;
   S702_BT_CODE_2105.RBT14_STANDARD_WELD_DATA := W#16#0;
   S702_BT_CODE_2105.RBT15_STANDARD_WELD_DATA := W#16#0;
   S702_BT_CODE_2105.RBT16_STANDARD_WELD_DATA := W#16#0;
   S702_BT_CODE_2105.RBT17_STANDARD_WELD_DATA := W#16#0;
   S702_BT_CODE_2105.RBT18_STANDARD_WELD_DATA := W#16#0;
   S702_BT_CODE_2105.RBT19_STANDARD_WELD_DATA := W#16#0;
   S702_BT_CODE_2105.RBT20_STANDARD_WELD_DATA := W#16#0;
   S702_BT_CODE_2105.RBT21_STANDARD_WELD_DATA := W#16#0;
   S702_BT_CODE_2105.RBT22_STANDARD_WELD_DATA := W#16#0;
   S702_BT_CODE_2105.RBT23_STANDARD_WELD_DAT := W#16#0;
   S702_BT_CODE_2105.RBT24_STANDARD_WELD_DAT := W#16#0;
   S702_BT_CODE_2105.CHK_WORD := W#16#0;
   S702_BT_CODE_2105.TEST_TEMP[1] := B#16#0;
   S702_BT_CODE_2105.TEST_TEMP[2] := B#16#0;
   S702_BT_CODE_2105.TEST_TEMP[3] := B#16#0;
   S702_BT_CODE_2105.TEST_TEMP[4] := B#16#0;
   S702_BT_CODE_2105.TEST_TEMP[5] := B#16#0;
   S702_BT_CODE_2105.TEST_TEMP[6] := B#16#0;
   S702_BT_CODE_2105.TEST_TEMP[7] := B#16#0;
   S702_BT_CODE_2105.TEST_TEMP[8] := B#16#0;
   S702_BT_CODE_2105.TEST_TEMP[9] := B#16#0;
   S702_BT_CODE_2105.TEST_TEMP[10] := B#16#0;
   S702_BT_CODE_2105.TEST_TEMP[11] := B#16#0;
   S702_BT_CODE_2105.TEST_TEMP[12] := B#16#0;
   S702_BT_CODE_2105.TEST_TEMP[13] := B#16#0;
   S702_BT_CODE_2105.TEST_TEMP[14] := B#16#0;
   S702_BT_CODE_2105.TEST_TEMP[15] := B#16#0;
   S702_BT_CODE_2105.TEST_TEMP[16] := B#16#0;
   S702_BT_CODE_2105.TEST_TEMP[17] := B#16#0;
   S702_BT_CODE_2105.TEST_TEMP[18] := B#16#0;
   S702_BT_CODE_2105.TEST_TEMP[19] := B#16#0;
   S702_BT_CODE_2105.TEST_TEMP[20] := B#16#0;
   S702_BT_CODE_2105.TEST_TEMP[21] := B#16#0;
   S702_BT_CODE_2105.TEST_TEMP[22] := B#16#0;
   S702_BT_CODE_2105.TEST_TEMP[23] := B#16#0;
   S702_BT_CODE_2105.TEST_TEMP[24] := B#16#0;
   S702_BT_CODE_2105.TEST_TEMP[25] := B#16#0;
   S702_BT_CODE_2105.TEST_TEMP[26] := B#16#0;
   S702_BT_CODE_2105.TEST_TEMP[27] := B#16#0;
   S702_BT_CODE_2105.TEST_TEMP[28] := B#16#0;
   S702_BT_CODE_2105.TEST_TEMP[29] := B#16#0;
   S702_BT_CODE_2105.TEST_TEMP[30] := B#16#0;
   S702_BT_CODE_2105.TEST_TEMP[31] := B#16#0;
   S702_BT_CODE_2105.TEST_TEMP[32] := B#16#0;
   S702_BT_CODE_2105.TEST_TEMP[33] := B#16#0;
   S702_BT_CODE_2105.TEST_TEMP[34] := B#16#0;
   S702_BT_CODE_2105.TEST_TEMP[35] := B#16#0;
   S702_BT_CODE_2105.TEST_TEMP[36] := B#16#0;
   S702_BT_CODE_2105.TEST_TEMP[37] := B#16#0;
   S702_BT_CODE_2105.TEST_TEMP[38] := B#16#0;
   S702_BT_CODE_2105.TEST_TEMP[39] := B#16#0;
   S702_BT_CODE_2105.TEST_TEMP[40] := B#16#0;
   S702_BT_CODE_2106.STATION_MAIN := W#16#0;
   S702_BT_CODE_2106.DISTINCTION_LH_RH := W#16#0;
   S702_BT_CODE_2106.STAION_NUMBER := W#16#0;
   S702_BT_CODE_2106.BODY_TYPE_1ST := W#16#0;
   S702_BT_CODE_2106.BODY_TYPE_OPTION := W#16#0;
   S702_BT_CODE_2106.RBT1_STANDARD_WELD_DATA := W#16#0;
   S702_BT_CODE_2106.RBT2_STANDARD_WELD_DATA := W#16#0;
   S702_BT_CODE_2106.RBT3_STANDARD_WELD_DATA := W#16#0;
   S702_BT_CODE_2106.RBT4_STANDARD_WELD_DATA := W#16#0;
   S702_BT_CODE_2106.RBT5_STANDARD_WELD_DATA := W#16#0;
   S702_BT_CODE_2106.RBT6_STANDARD_WELD_DATA := W#16#0;
   S702_BT_CODE_2106.RBT7_STANDARD_WELD_DATA := W#16#0;
   S702_BT_CODE_2106.RBT8_STANDARD_WELD_DATA := W#16#0;
   S702_BT_CODE_2106.RBT9_STANDARD_WELD_DATA := W#16#0;
   S702_BT_CODE_2106.RBT10_STANDARD_WELD_DATA := W#16#0;
   S702_BT_CODE_2106.RBT11_STANDARD_WELD_DATA := W#16#0;
   S702_BT_CODE_2106.RBT12_STANDARD_WELD_DATA := W#16#0;
   S702_BT_CODE_2106.RBT13_STANDARD_WELD_DATA := W#16#0;
   S702_BT_CODE_2106.RBT14_STANDARD_WELD_DATA := W#16#0;
   S702_BT_CODE_2106.RBT15_STANDARD_WELD_DATA := W#16#0;
   S702_BT_CODE_2106.RBT16_STANDARD_WELD_DATA := W#16#0;
   S702_BT_CODE_2106.RBT17_STANDARD_WELD_DATA := W#16#0;
   S702_BT_CODE_2106.RBT18_STANDARD_WELD_DATA := W#16#0;
   S702_BT_CODE_2106.RBT19_STANDARD_WELD_DATA := W#16#0;
   S702_BT_CODE_2106.RBT20_STANDARD_WELD_DATA := W#16#0;
   S702_BT_CODE_2106.RBT21_STANDARD_WELD_DATA := W#16#0;
   S702_BT_CODE_2106.RBT22_STANDARD_WELD_DATA := W#16#0;
   S702_BT_CODE_2106.RBT23_STANDARD_WELD_DAT := W#16#0;
   S702_BT_CODE_2106.RBT24_STANDARD_WELD_DAT := W#16#0;
   S702_BT_CODE_2106.CHK_WORD := W#16#0;
   S702_BT_CODE_2106.TEST_TEMP[1] := B#16#0;
   S702_BT_CODE_2106.TEST_TEMP[2] := B#16#0;
   S702_BT_CODE_2106.TEST_TEMP[3] := B#16#0;
   S702_BT_CODE_2106.TEST_TEMP[4] := B#16#0;
   S702_BT_CODE_2106.TEST_TEMP[5] := B#16#0;
   S702_BT_CODE_2106.TEST_TEMP[6] := B#16#0;
   S702_BT_CODE_2106.TEST_TEMP[7] := B#16#0;
   S702_BT_CODE_2106.TEST_TEMP[8] := B#16#0;
   S702_BT_CODE_2106.TEST_TEMP[9] := B#16#0;
   S702_BT_CODE_2106.TEST_TEMP[10] := B#16#0;
   S702_BT_CODE_2106.TEST_TEMP[11] := B#16#0;
   S702_BT_CODE_2106.TEST_TEMP[12] := B#16#0;
   S702_BT_CODE_2106.TEST_TEMP[13] := B#16#0;
   S702_BT_CODE_2106.TEST_TEMP[14] := B#16#0;
   S702_BT_CODE_2106.TEST_TEMP[15] := B#16#0;
   S702_BT_CODE_2106.TEST_TEMP[16] := B#16#0;
   S702_BT_CODE_2106.TEST_TEMP[17] := B#16#0;
   S702_BT_CODE_2106.TEST_TEMP[18] := B#16#0;
   S702_BT_CODE_2106.TEST_TEMP[19] := B#16#0;
   S702_BT_CODE_2106.TEST_TEMP[20] := B#16#0;
   S702_BT_CODE_2106.TEST_TEMP[21] := B#16#0;
   S702_BT_CODE_2106.TEST_TEMP[22] := B#16#0;
   S702_BT_CODE_2106.TEST_TEMP[23] := B#16#0;
   S702_BT_CODE_2106.TEST_TEMP[24] := B#16#0;
   S702_BT_CODE_2106.TEST_TEMP[25] := B#16#0;
   S702_BT_CODE_2106.TEST_TEMP[26] := B#16#0;
   S702_BT_CODE_2106.TEST_TEMP[27] := B#16#0;
   S702_BT_CODE_2106.TEST_TEMP[28] := B#16#0;
   S702_BT_CODE_2106.TEST_TEMP[29] := B#16#0;
   S702_BT_CODE_2106.TEST_TEMP[30] := B#16#0;
   S702_BT_CODE_2106.TEST_TEMP[31] := B#16#0;
   S702_BT_CODE_2106.TEST_TEMP[32] := B#16#0;
   S702_BT_CODE_2106.TEST_TEMP[33] := B#16#0;
   S702_BT_CODE_2106.TEST_TEMP[34] := B#16#0;
   S702_BT_CODE_2106.TEST_TEMP[35] := B#16#0;
   S702_BT_CODE_2106.TEST_TEMP[36] := B#16#0;
   S702_BT_CODE_2106.TEST_TEMP[37] := B#16#0;
   S702_BT_CODE_2106.TEST_TEMP[38] := B#16#0;
   S702_BT_CODE_2106.TEST_TEMP[39] := B#16#0;
   S702_BT_CODE_2106.TEST_TEMP[40] := B#16#0;
   S702_BT_CODE_2107.STATION_MAIN := W#16#0;
   S702_BT_CODE_2107.DISTINCTION_LH_RH := W#16#0;
   S702_BT_CODE_2107.STAION_NUMBER := W#16#0;
   S702_BT_CODE_2107.BODY_TYPE_1ST := W#16#0;
   S702_BT_CODE_2107.BODY_TYPE_OPTION := W#16#0;
   S702_BT_CODE_2107.RBT1_STANDARD_WELD_DATA := W#16#0;
   S702_BT_CODE_2107.RBT2_STANDARD_WELD_DATA := W#16#0;
   S702_BT_CODE_2107.RBT3_STANDARD_WELD_DATA := W#16#0;
   S702_BT_CODE_2107.RBT4_STANDARD_WELD_DATA := W#16#0;
   S702_BT_CODE_2107.RBT5_STANDARD_WELD_DATA := W#16#0;
   S702_BT_CODE_2107.RBT6_STANDARD_WELD_DATA := W#16#0;
   S702_BT_CODE_2107.RBT7_STANDARD_WELD_DATA := W#16#0;
   S702_BT_CODE_2107.RBT8_STANDARD_WELD_DATA := W#16#0;
   S702_BT_CODE_2107.RBT9_STANDARD_WELD_DATA := W#16#0;
   S702_BT_CODE_2107.RBT10_STANDARD_WELD_DATA := W#16#0;
   S702_BT_CODE_2107.RBT11_STANDARD_WELD_DATA := W#16#0;
   S702_BT_CODE_2107.RBT12_STANDARD_WELD_DATA := W#16#0;
   S702_BT_CODE_2107.RBT13_STANDARD_WELD_DATA := W#16#0;
   S702_BT_CODE_2107.RBT14_STANDARD_WELD_DATA := W#16#0;
   S702_BT_CODE_2107.RBT15_STANDARD_WELD_DATA := W#16#0;
   S702_BT_CODE_2107.RBT16_STANDARD_WELD_DATA := W#16#0;
   S702_BT_CODE_2107.RBT17_STANDARD_WELD_DATA := W#16#0;
   S702_BT_CODE_2107.RBT18_STANDARD_WELD_DATA := W#16#0;
   S702_BT_CODE_2107.RBT19_STANDARD_WELD_DATA := W#16#0;
   S702_BT_CODE_2107.RBT20_STANDARD_WELD_DATA := W#16#0;
   S702_BT_CODE_2107.RBT21_STANDARD_WELD_DATA := W#16#0;
   S702_BT_CODE_2107.RBT22_STANDARD_WELD_DATA := W#16#0;
   S702_BT_CODE_2107.RBT23_STANDARD_WELD_DAT := W#16#0;
   S702_BT_CODE_2107.RBT24_STANDARD_WELD_DAT := W#16#0;
   S702_BT_CODE_2107.CHK_WORD := W#16#0;
   S702_BT_CODE_2107.TEST_TEMP[1] := B#16#0;
   S702_BT_CODE_2107.TEST_TEMP[2] := B#16#0;
   S702_BT_CODE_2107.TEST_TEMP[3] := B#16#0;
   S702_BT_CODE_2107.TEST_TEMP[4] := B#16#0;
   S702_BT_CODE_2107.TEST_TEMP[5] := B#16#0;
   S702_BT_CODE_2107.TEST_TEMP[6] := B#16#0;
   S702_BT_CODE_2107.TEST_TEMP[7] := B#16#0;
   S702_BT_CODE_2107.TEST_TEMP[8] := B#16#0;
   S702_BT_CODE_2107.TEST_TEMP[9] := B#16#0;
   S702_BT_CODE_2107.TEST_TEMP[10] := B#16#0;
   S702_BT_CODE_2107.TEST_TEMP[11] := B#16#0;
   S702_BT_CODE_2107.TEST_TEMP[12] := B#16#0;
   S702_BT_CODE_2107.TEST_TEMP[13] := B#16#0;
   S702_BT_CODE_2107.TEST_TEMP[14] := B#16#0;
   S702_BT_CODE_2107.TEST_TEMP[15] := B#16#0;
   S702_BT_CODE_2107.TEST_TEMP[16] := B#16#0;
   S702_BT_CODE_2107.TEST_TEMP[17] := B#16#0;
   S702_BT_CODE_2107.TEST_TEMP[18] := B#16#0;
   S702_BT_CODE_2107.TEST_TEMP[19] := B#16#0;
   S702_BT_CODE_2107.TEST_TEMP[20] := B#16#0;
   S702_BT_CODE_2107.TEST_TEMP[21] := B#16#0;
   S702_BT_CODE_2107.TEST_TEMP[22] := B#16#0;
   S702_BT_CODE_2107.TEST_TEMP[23] := B#16#0;
   S702_BT_CODE_2107.TEST_TEMP[24] := B#16#0;
   S702_BT_CODE_2107.TEST_TEMP[25] := B#16#0;
   S702_BT_CODE_2107.TEST_TEMP[26] := B#16#0;
   S702_BT_CODE_2107.TEST_TEMP[27] := B#16#0;
   S702_BT_CODE_2107.TEST_TEMP[28] := B#16#0;
   S702_BT_CODE_2107.TEST_TEMP[29] := B#16#0;
   S702_BT_CODE_2107.TEST_TEMP[30] := B#16#0;
   S702_BT_CODE_2107.TEST_TEMP[31] := B#16#0;
   S702_BT_CODE_2107.TEST_TEMP[32] := B#16#0;
   S702_BT_CODE_2107.TEST_TEMP[33] := B#16#0;
   S702_BT_CODE_2107.TEST_TEMP[34] := B#16#0;
   S702_BT_CODE_2107.TEST_TEMP[35] := B#16#0;
   S702_BT_CODE_2107.TEST_TEMP[36] := B#16#0;
   S702_BT_CODE_2107.TEST_TEMP[37] := B#16#0;
   S702_BT_CODE_2107.TEST_TEMP[38] := B#16#0;
   S702_BT_CODE_2107.TEST_TEMP[39] := B#16#0;
   S702_BT_CODE_2107.TEST_TEMP[40] := B#16#0;
   S702_BT_CODE_2108.STATION_MAIN := W#16#0;
   S702_BT_CODE_2108.DISTINCTION_LH_RH := W#16#0;
   S702_BT_CODE_2108.STAION_NUMBER := W#16#0;
   S702_BT_CODE_2108.BODY_TYPE_1ST := W#16#0;
   S702_BT_CODE_2108.BODY_TYPE_OPTION := W#16#0;
   S702_BT_CODE_2108.RBT1_STANDARD_WELD_DATA := W#16#0;
   S702_BT_CODE_2108.RBT2_STANDARD_WELD_DATA := W#16#0;
   S702_BT_CODE_2108.RBT3_STANDARD_WELD_DATA := W#16#0;
   S702_BT_CODE_2108.RBT4_STANDARD_WELD_DATA := W#16#0;
   S702_BT_CODE_2108.RBT5_STANDARD_WELD_DATA := W#16#0;
   S702_BT_CODE_2108.RBT6_STANDARD_WELD_DATA := W#16#0;
   S702_BT_CODE_2108.RBT7_STANDARD_WELD_DATA := W#16#0;
   S702_BT_CODE_2108.RBT8_STANDARD_WELD_DATA := W#16#0;
   S702_BT_CODE_2108.RBT9_STANDARD_WELD_DATA := W#16#0;
   S702_BT_CODE_2108.RBT10_STANDARD_WELD_DATA := W#16#0;
   S702_BT_CODE_2108.RBT11_STANDARD_WELD_DATA := W#16#0;
   S702_BT_CODE_2108.RBT12_STANDARD_WELD_DATA := W#16#0;
   S702_BT_CODE_2108.RBT13_STANDARD_WELD_DATA := W#16#0;
   S702_BT_CODE_2108.RBT14_STANDARD_WELD_DATA := W#16#0;
   S702_BT_CODE_2108.RBT15_STANDARD_WELD_DATA := W#16#0;
   S702_BT_CODE_2108.RBT16_STANDARD_WELD_DATA := W#16#0;
   S702_BT_CODE_2108.RBT17_STANDARD_WELD_DATA := W#16#0;
   S702_BT_CODE_2108.RBT18_STANDARD_WELD_DATA := W#16#0;
   S702_BT_CODE_2108.RBT19_STANDARD_WELD_DATA := W#16#0;
   S702_BT_CODE_2108.RBT20_STANDARD_WELD_DATA := W#16#0;
   S702_BT_CODE_2108.RBT21_STANDARD_WELD_DATA := W#16#0;
   S702_BT_CODE_2108.RBT22_STANDARD_WELD_DATA := W#16#0;
   S702_BT_CODE_2108.RBT23_STANDARD_WELD_DAT := W#16#0;
   S702_BT_CODE_2108.RBT24_STANDARD_WELD_DAT := W#16#0;
   S702_BT_CODE_2108.CHK_WORD := W#16#0;
   S702_BT_CODE_2108.TEST_TEMP[1] := B#16#0;
   S702_BT_CODE_2108.TEST_TEMP[2] := B#16#0;
   S702_BT_CODE_2108.TEST_TEMP[3] := B#16#0;
   S702_BT_CODE_2108.TEST_TEMP[4] := B#16#0;
   S702_BT_CODE_2108.TEST_TEMP[5] := B#16#0;
   S702_BT_CODE_2108.TEST_TEMP[6] := B#16#0;
   S702_BT_CODE_2108.TEST_TEMP[7] := B#16#0;
   S702_BT_CODE_2108.TEST_TEMP[8] := B#16#0;
   S702_BT_CODE_2108.TEST_TEMP[9] := B#16#0;
   S702_BT_CODE_2108.TEST_TEMP[10] := B#16#0;
   S702_BT_CODE_2108.TEST_TEMP[11] := B#16#0;
   S702_BT_CODE_2108.TEST_TEMP[12] := B#16#0;
   S702_BT_CODE_2108.TEST_TEMP[13] := B#16#0;
   S702_BT_CODE_2108.TEST_TEMP[14] := B#16#0;
   S702_BT_CODE_2108.TEST_TEMP[15] := B#16#0;
   S702_BT_CODE_2108.TEST_TEMP[16] := B#16#0;
   S702_BT_CODE_2108.TEST_TEMP[17] := B#16#0;
   S702_BT_CODE_2108.TEST_TEMP[18] := B#16#0;
   S702_BT_CODE_2108.TEST_TEMP[19] := B#16#0;
   S702_BT_CODE_2108.TEST_TEMP[20] := B#16#0;
   S702_BT_CODE_2108.TEST_TEMP[21] := B#16#0;
   S702_BT_CODE_2108.TEST_TEMP[22] := B#16#0;
   S702_BT_CODE_2108.TEST_TEMP[23] := B#16#0;
   S702_BT_CODE_2108.TEST_TEMP[24] := B#16#0;
   S702_BT_CODE_2108.TEST_TEMP[25] := B#16#0;
   S702_BT_CODE_2108.TEST_TEMP[26] := B#16#0;
   S702_BT_CODE_2108.TEST_TEMP[27] := B#16#0;
   S702_BT_CODE_2108.TEST_TEMP[28] := B#16#0;
   S702_BT_CODE_2108.TEST_TEMP[29] := B#16#0;
   S702_BT_CODE_2108.TEST_TEMP[30] := B#16#0;
   S702_BT_CODE_2108.TEST_TEMP[31] := B#16#0;
   S702_BT_CODE_2108.TEST_TEMP[32] := B#16#0;
   S702_BT_CODE_2108.TEST_TEMP[33] := B#16#0;
   S702_BT_CODE_2108.TEST_TEMP[34] := B#16#0;
   S702_BT_CODE_2108.TEST_TEMP[35] := B#16#0;
   S702_BT_CODE_2108.TEST_TEMP[36] := B#16#0;
   S702_BT_CODE_2108.TEST_TEMP[37] := B#16#0;
   S702_BT_CODE_2108.TEST_TEMP[38] := B#16#0;
   S702_BT_CODE_2108.TEST_TEMP[39] := B#16#0;
   S702_BT_CODE_2108.TEST_TEMP[40] := B#16#0;
   S702_BT_CODE_2109.STATION_MAIN := W#16#0;
   S702_BT_CODE_2109.DISTINCTION_LH_RH := W#16#0;
   S702_BT_CODE_2109.STAION_NUMBER := W#16#0;
   S702_BT_CODE_2109.BODY_TYPE_1ST := W#16#0;
   S702_BT_CODE_2109.BODY_TYPE_OPTION := W#16#0;
   S702_BT_CODE_2109.RBT1_STANDARD_WELD_DATA := W#16#0;
   S702_BT_CODE_2109.RBT2_STANDARD_WELD_DATA := W#16#0;
   S702_BT_CODE_2109.RBT3_STANDARD_WELD_DATA := W#16#0;
   S702_BT_CODE_2109.RBT4_STANDARD_WELD_DATA := W#16#0;
   S702_BT_CODE_2109.RBT5_STANDARD_WELD_DATA := W#16#0;
   S702_BT_CODE_2109.RBT6_STANDARD_WELD_DATA := W#16#0;
   S702_BT_CODE_2109.RBT7_STANDARD_WELD_DATA := W#16#0;
   S702_BT_CODE_2109.RBT8_STANDARD_WELD_DATA := W#16#0;
   S702_BT_CODE_2109.RBT9_STANDARD_WELD_DATA := W#16#0;
   S702_BT_CODE_2109.RBT10_STANDARD_WELD_DATA := W#16#0;
   S702_BT_CODE_2109.RBT11_STANDARD_WELD_DATA := W#16#0;
   S702_BT_CODE_2109.RBT12_STANDARD_WELD_DATA := W#16#0;
   S702_BT_CODE_2109.RBT13_STANDARD_WELD_DATA := W#16#0;
   S702_BT_CODE_2109.RBT14_STANDARD_WELD_DATA := W#16#0;
   S702_BT_CODE_2109.RBT15_STANDARD_WELD_DATA := W#16#0;
   S702_BT_CODE_2109.RBT16_STANDARD_WELD_DATA := W#16#0;
   S702_BT_CODE_2109.RBT17_STANDARD_WELD_DATA := W#16#0;
   S702_BT_CODE_2109.RBT18_STANDARD_WELD_DATA := W#16#0;
   S702_BT_CODE_2109.RBT19_STANDARD_WELD_DATA := W#16#0;
   S702_BT_CODE_2109.RBT20_STANDARD_WELD_DATA := W#16#0;
   S702_BT_CODE_2109.RBT21_STANDARD_WELD_DATA := W#16#0;
   S702_BT_CODE_2109.RBT22_STANDARD_WELD_DATA := W#16#0;
   S702_BT_CODE_2109.RBT23_STANDARD_WELD_DAT := W#16#0;
   S702_BT_CODE_2109.RBT24_STANDARD_WELD_DAT := W#16#0;
   S702_BT_CODE_2109.CHK_WORD := W#16#0;
   S702_BT_CODE_2109.TEST_TEMP[1] := B#16#0;
   S702_BT_CODE_2109.TEST_TEMP[2] := B#16#0;
   S702_BT_CODE_2109.TEST_TEMP[3] := B#16#0;
   S702_BT_CODE_2109.TEST_TEMP[4] := B#16#0;
   S702_BT_CODE_2109.TEST_TEMP[5] := B#16#0;
   S702_BT_CODE_2109.TEST_TEMP[6] := B#16#0;
   S702_BT_CODE_2109.TEST_TEMP[7] := B#16#0;
   S702_BT_CODE_2109.TEST_TEMP[8] := B#16#0;
   S702_BT_CODE_2109.TEST_TEMP[9] := B#16#0;
   S702_BT_CODE_2109.TEST_TEMP[10] := B#16#0;
   S702_BT_CODE_2109.TEST_TEMP[11] := B#16#0;
   S702_BT_CODE_2109.TEST_TEMP[12] := B#16#0;
   S702_BT_CODE_2109.TEST_TEMP[13] := B#16#0;
   S702_BT_CODE_2109.TEST_TEMP[14] := B#16#0;
   S702_BT_CODE_2109.TEST_TEMP[15] := B#16#0;
   S702_BT_CODE_2109.TEST_TEMP[16] := B#16#0;
   S702_BT_CODE_2109.TEST_TEMP[17] := B#16#0;
   S702_BT_CODE_2109.TEST_TEMP[18] := B#16#0;
   S702_BT_CODE_2109.TEST_TEMP[19] := B#16#0;
   S702_BT_CODE_2109.TEST_TEMP[20] := B#16#0;
   S702_BT_CODE_2109.TEST_TEMP[21] := B#16#0;
   S702_BT_CODE_2109.TEST_TEMP[22] := B#16#0;
   S702_BT_CODE_2109.TEST_TEMP[23] := B#16#0;
   S702_BT_CODE_2109.TEST_TEMP[24] := B#16#0;
   S702_BT_CODE_2109.TEST_TEMP[25] := B#16#0;
   S702_BT_CODE_2109.TEST_TEMP[26] := B#16#0;
   S702_BT_CODE_2109.TEST_TEMP[27] := B#16#0;
   S702_BT_CODE_2109.TEST_TEMP[28] := B#16#0;
   S702_BT_CODE_2109.TEST_TEMP[29] := B#16#0;
   S702_BT_CODE_2109.TEST_TEMP[30] := B#16#0;
   S702_BT_CODE_2109.TEST_TEMP[31] := B#16#0;
   S702_BT_CODE_2109.TEST_TEMP[32] := B#16#0;
   S702_BT_CODE_2109.TEST_TEMP[33] := B#16#0;
   S702_BT_CODE_2109.TEST_TEMP[34] := B#16#0;
   S702_BT_CODE_2109.TEST_TEMP[35] := B#16#0;
   S702_BT_CODE_2109.TEST_TEMP[36] := B#16#0;
   S702_BT_CODE_2109.TEST_TEMP[37] := B#16#0;
   S702_BT_CODE_2109.TEST_TEMP[38] := B#16#0;
   S702_BT_CODE_2109.TEST_TEMP[39] := B#16#0;
   S702_BT_CODE_2109.TEST_TEMP[40] := B#16#0;
   S702_BT_CODE_2110.STATION_MAIN := W#16#0;
   S702_BT_CODE_2110.DISTINCTION_LH_RH := W#16#0;
   S702_BT_CODE_2110.STAION_NUMBER := W#16#0;
   S702_BT_CODE_2110.BODY_TYPE_1ST := W#16#0;
   S702_BT_CODE_2110.BODY_TYPE_OPTION := W#16#0;
   S702_BT_CODE_2110.RBT1_STANDARD_WELD_DATA := W#16#0;
   S702_BT_CODE_2110.RBT2_STANDARD_WELD_DATA := W#16#0;
   S702_BT_CODE_2110.RBT3_STANDARD_WELD_DATA := W#16#0;
   S702_BT_CODE_2110.RBT4_STANDARD_WELD_DATA := W#16#0;
   S702_BT_CODE_2110.RBT5_STANDARD_WELD_DATA := W#16#0;
   S702_BT_CODE_2110.RBT6_STANDARD_WELD_DATA := W#16#0;
   S702_BT_CODE_2110.RBT7_STANDARD_WELD_DATA := W#16#0;
   S702_BT_CODE_2110.RBT8_STANDARD_WELD_DATA := W#16#0;
   S702_BT_CODE_2110.RBT9_STANDARD_WELD_DATA := W#16#0;
   S702_BT_CODE_2110.RBT10_STANDARD_WELD_DATA := W#16#0;
   S702_BT_CODE_2110.RBT11_STANDARD_WELD_DATA := W#16#0;
   S702_BT_CODE_2110.RBT12_STANDARD_WELD_DATA := W#16#0;
   S702_BT_CODE_2110.RBT13_STANDARD_WELD_DATA := W#16#0;
   S702_BT_CODE_2110.RBT14_STANDARD_WELD_DATA := W#16#0;
   S702_BT_CODE_2110.RBT15_STANDARD_WELD_DATA := W#16#0;
   S702_BT_CODE_2110.RBT16_STANDARD_WELD_DATA := W#16#0;
   S702_BT_CODE_2110.RBT17_STANDARD_WELD_DATA := W#16#0;
   S702_BT_CODE_2110.RBT18_STANDARD_WELD_DATA := W#16#0;
   S702_BT_CODE_2110.RBT19_STANDARD_WELD_DATA := W#16#0;
   S702_BT_CODE_2110.RBT20_STANDARD_WELD_DATA := W#16#0;
   S702_BT_CODE_2110.RBT21_STANDARD_WELD_DATA := W#16#0;
   S702_BT_CODE_2110.RBT22_STANDARD_WELD_DATA := W#16#0;
   S702_BT_CODE_2110.RBT23_STANDARD_WELD_DAT := W#16#0;
   S702_BT_CODE_2110.RBT24_STANDARD_WELD_DAT := W#16#0;
   S702_BT_CODE_2110.CHK_WORD := W#16#0;
   S702_BT_CODE_2110.TEST_TEMP[1] := B#16#0;
   S702_BT_CODE_2110.TEST_TEMP[2] := B#16#0;
   S702_BT_CODE_2110.TEST_TEMP[3] := B#16#0;
   S702_BT_CODE_2110.TEST_TEMP[4] := B#16#0;
   S702_BT_CODE_2110.TEST_TEMP[5] := B#16#0;
   S702_BT_CODE_2110.TEST_TEMP[6] := B#16#0;
   S702_BT_CODE_2110.TEST_TEMP[7] := B#16#0;
   S702_BT_CODE_2110.TEST_TEMP[8] := B#16#0;
   S702_BT_CODE_2110.TEST_TEMP[9] := B#16#0;
   S702_BT_CODE_2110.TEST_TEMP[10] := B#16#0;
   S702_BT_CODE_2110.TEST_TEMP[11] := B#16#0;
   S702_BT_CODE_2110.TEST_TEMP[12] := B#16#0;
   S702_BT_CODE_2110.TEST_TEMP[13] := B#16#0;
   S702_BT_CODE_2110.TEST_TEMP[14] := B#16#0;
   S702_BT_CODE_2110.TEST_TEMP[15] := B#16#0;
   S702_BT_CODE_2110.TEST_TEMP[16] := B#16#0;
   S702_BT_CODE_2110.TEST_TEMP[17] := B#16#0;
   S702_BT_CODE_2110.TEST_TEMP[18] := B#16#0;
   S702_BT_CODE_2110.TEST_TEMP[19] := B#16#0;
   S702_BT_CODE_2110.TEST_TEMP[20] := B#16#0;
   S702_BT_CODE_2110.TEST_TEMP[21] := B#16#0;
   S702_BT_CODE_2110.TEST_TEMP[22] := B#16#0;
   S702_BT_CODE_2110.TEST_TEMP[23] := B#16#0;
   S702_BT_CODE_2110.TEST_TEMP[24] := B#16#0;
   S702_BT_CODE_2110.TEST_TEMP[25] := B#16#0;
   S702_BT_CODE_2110.TEST_TEMP[26] := B#16#0;
   S702_BT_CODE_2110.TEST_TEMP[27] := B#16#0;
   S702_BT_CODE_2110.TEST_TEMP[28] := B#16#0;
   S702_BT_CODE_2110.TEST_TEMP[29] := B#16#0;
   S702_BT_CODE_2110.TEST_TEMP[30] := B#16#0;
   S702_BT_CODE_2110.TEST_TEMP[31] := B#16#0;
   S702_BT_CODE_2110.TEST_TEMP[32] := B#16#0;
   S702_BT_CODE_2110.TEST_TEMP[33] := B#16#0;
   S702_BT_CODE_2110.TEST_TEMP[34] := B#16#0;
   S702_BT_CODE_2110.TEST_TEMP[35] := B#16#0;
   S702_BT_CODE_2110.TEST_TEMP[36] := B#16#0;
   S702_BT_CODE_2110.TEST_TEMP[37] := B#16#0;
   S702_BT_CODE_2110.TEST_TEMP[38] := B#16#0;
   S702_BT_CODE_2110.TEST_TEMP[39] := B#16#0;
   S702_BT_CODE_2110.TEST_TEMP[40] := B#16#0;
   S702_BT_CODE_2111.STATION_MAIN := W#16#0;
   S702_BT_CODE_2111.DISTINCTION_LH_RH := W#16#0;
   S702_BT_CODE_2111.STAION_NUMBER := W#16#0;
   S702_BT_CODE_2111.BODY_TYPE_1ST := W#16#0;
   S702_BT_CODE_2111.BODY_TYPE_OPTION := W#16#0;
   S702_BT_CODE_2111.RBT1_STANDARD_WELD_DATA := W#16#0;
   S702_BT_CODE_2111.RBT2_STANDARD_WELD_DATA := W#16#0;
   S702_BT_CODE_2111.RBT3_STANDARD_WELD_DATA := W#16#0;
   S702_BT_CODE_2111.RBT4_STANDARD_WELD_DATA := W#16#0;
   S702_BT_CODE_2111.RBT5_STANDARD_WELD_DATA := W#16#0;
   S702_BT_CODE_2111.RBT6_STANDARD_WELD_DATA := W#16#0;
   S702_BT_CODE_2111.RBT7_STANDARD_WELD_DATA := W#16#0;
   S702_BT_CODE_2111.RBT8_STANDARD_WELD_DATA := W#16#0;
   S702_BT_CODE_2111.RBT9_STANDARD_WELD_DATA := W#16#0;
   S702_BT_CODE_2111.RBT10_STANDARD_WELD_DATA := W#16#0;
   S702_BT_CODE_2111.RBT11_STANDARD_WELD_DATA := W#16#0;
   S702_BT_CODE_2111.RBT12_STANDARD_WELD_DATA := W#16#0;
   S702_BT_CODE_2111.RBT13_STANDARD_WELD_DATA := W#16#0;
   S702_BT_CODE_2111.RBT14_STANDARD_WELD_DATA := W#16#0;
   S702_BT_CODE_2111.RBT15_STANDARD_WELD_DATA := W#16#0;
   S702_BT_CODE_2111.RBT16_STANDARD_WELD_DATA := W#16#0;
   S702_BT_CODE_2111.RBT17_STANDARD_WELD_DATA := W#16#0;
   S702_BT_CODE_2111.RBT18_STANDARD_WELD_DATA := W#16#0;
   S702_BT_CODE_2111.RBT19_STANDARD_WELD_DATA := W#16#0;
   S702_BT_CODE_2111.RBT20_STANDARD_WELD_DATA := W#16#0;
   S702_BT_CODE_2111.RBT21_STANDARD_WELD_DATA := W#16#0;
   S702_BT_CODE_2111.RBT22_STANDARD_WELD_DATA := W#16#0;
   S702_BT_CODE_2111.RBT23_STANDARD_WELD_DAT := W#16#0;
   S702_BT_CODE_2111.RBT24_STANDARD_WELD_DAT := W#16#0;
   S702_BT_CODE_2111.CHK_WORD := W#16#0;
   S702_BT_CODE_2111.TEST_TEMP[1] := B#16#0;
   S702_BT_CODE_2111.TEST_TEMP[2] := B#16#0;
   S702_BT_CODE_2111.TEST_TEMP[3] := B#16#0;
   S702_BT_CODE_2111.TEST_TEMP[4] := B#16#0;
   S702_BT_CODE_2111.TEST_TEMP[5] := B#16#0;
   S702_BT_CODE_2111.TEST_TEMP[6] := B#16#0;
   S702_BT_CODE_2111.TEST_TEMP[7] := B#16#0;
   S702_BT_CODE_2111.TEST_TEMP[8] := B#16#0;
   S702_BT_CODE_2111.TEST_TEMP[9] := B#16#0;
   S702_BT_CODE_2111.TEST_TEMP[10] := B#16#0;
   S702_BT_CODE_2111.TEST_TEMP[11] := B#16#0;
   S702_BT_CODE_2111.TEST_TEMP[12] := B#16#0;
   S702_BT_CODE_2111.TEST_TEMP[13] := B#16#0;
   S702_BT_CODE_2111.TEST_TEMP[14] := B#16#0;
   S702_BT_CODE_2111.TEST_TEMP[15] := B#16#0;
   S702_BT_CODE_2111.TEST_TEMP[16] := B#16#0;
   S702_BT_CODE_2111.TEST_TEMP[17] := B#16#0;
   S702_BT_CODE_2111.TEST_TEMP[18] := B#16#0;
   S702_BT_CODE_2111.TEST_TEMP[19] := B#16#0;
   S702_BT_CODE_2111.TEST_TEMP[20] := B#16#0;
   S702_BT_CODE_2111.TEST_TEMP[21] := B#16#0;
   S702_BT_CODE_2111.TEST_TEMP[22] := B#16#0;
   S702_BT_CODE_2111.TEST_TEMP[23] := B#16#0;
   S702_BT_CODE_2111.TEST_TEMP[24] := B#16#0;
   S702_BT_CODE_2111.TEST_TEMP[25] := B#16#0;
   S702_BT_CODE_2111.TEST_TEMP[26] := B#16#0;
   S702_BT_CODE_2111.TEST_TEMP[27] := B#16#0;
   S702_BT_CODE_2111.TEST_TEMP[28] := B#16#0;
   S702_BT_CODE_2111.TEST_TEMP[29] := B#16#0;
   S702_BT_CODE_2111.TEST_TEMP[30] := B#16#0;
   S702_BT_CODE_2111.TEST_TEMP[31] := B#16#0;
   S702_BT_CODE_2111.TEST_TEMP[32] := B#16#0;
   S702_BT_CODE_2111.TEST_TEMP[33] := B#16#0;
   S702_BT_CODE_2111.TEST_TEMP[34] := B#16#0;
   S702_BT_CODE_2111.TEST_TEMP[35] := B#16#0;
   S702_BT_CODE_2111.TEST_TEMP[36] := B#16#0;
   S702_BT_CODE_2111.TEST_TEMP[37] := B#16#0;
   S702_BT_CODE_2111.TEST_TEMP[38] := B#16#0;
   S702_BT_CODE_2111.TEST_TEMP[39] := B#16#0;
   S702_BT_CODE_2111.TEST_TEMP[40] := B#16#0;
   S702_BT_CODE_2112.STATION_MAIN := W#16#0;
   S702_BT_CODE_2112.DISTINCTION_LH_RH := W#16#0;
   S702_BT_CODE_2112.STAION_NUMBER := W#16#0;
   S702_BT_CODE_2112.BODY_TYPE_1ST := W#16#0;
   S702_BT_CODE_2112.BODY_TYPE_OPTION := W#16#0;
   S702_BT_CODE_2112.RBT1_STANDARD_WELD_DATA := W#16#0;
   S702_BT_CODE_2112.RBT2_STANDARD_WELD_DATA := W#16#0;
   S702_BT_CODE_2112.RBT3_STANDARD_WELD_DATA := W#16#0;
   S702_BT_CODE_2112.RBT4_STANDARD_WELD_DATA := W#16#0;
   S702_BT_CODE_2112.RBT5_STANDARD_WELD_DATA := W#16#0;
   S702_BT_CODE_2112.RBT6_STANDARD_WELD_DATA := W#16#0;
   S702_BT_CODE_2112.RBT7_STANDARD_WELD_DATA := W#16#0;
   S702_BT_CODE_2112.RBT8_STANDARD_WELD_DATA := W#16#0;
   S702_BT_CODE_2112.RBT9_STANDARD_WELD_DATA := W#16#0;
   S702_BT_CODE_2112.RBT10_STANDARD_WELD_DATA := W#16#0;
   S702_BT_CODE_2112.RBT11_STANDARD_WELD_DATA := W#16#0;
   S702_BT_CODE_2112.RBT12_STANDARD_WELD_DATA := W#16#0;
   S702_BT_CODE_2112.RBT13_STANDARD_WELD_DATA := W#16#0;
   S702_BT_CODE_2112.RBT14_STANDARD_WELD_DATA := W#16#0;
   S702_BT_CODE_2112.RBT15_STANDARD_WELD_DATA := W#16#0;
   S702_BT_CODE_2112.RBT16_STANDARD_WELD_DATA := W#16#0;
   S702_BT_CODE_2112.RBT17_STANDARD_WELD_DATA := W#16#0;
   S702_BT_CODE_2112.RBT18_STANDARD_WELD_DATA := W#16#0;
   S702_BT_CODE_2112.RBT19_STANDARD_WELD_DATA := W#16#0;
   S702_BT_CODE_2112.RBT20_STANDARD_WELD_DATA := W#16#0;
   S702_BT_CODE_2112.RBT21_STANDARD_WELD_DATA := W#16#0;
   S702_BT_CODE_2112.RBT22_STANDARD_WELD_DATA := W#16#0;
   S702_BT_CODE_2112.RBT23_STANDARD_WELD_DAT := W#16#0;
   S702_BT_CODE_2112.RBT24_STANDARD_WELD_DAT := W#16#0;
   S702_BT_CODE_2112.CHK_WORD := W#16#0;
   S702_BT_CODE_2112.TEST_TEMP[1] := B#16#0;
   S702_BT_CODE_2112.TEST_TEMP[2] := B#16#0;
   S702_BT_CODE_2112.TEST_TEMP[3] := B#16#0;
   S702_BT_CODE_2112.TEST_TEMP[4] := B#16#0;
   S702_BT_CODE_2112.TEST_TEMP[5] := B#16#0;
   S702_BT_CODE_2112.TEST_TEMP[6] := B#16#0;
   S702_BT_CODE_2112.TEST_TEMP[7] := B#16#0;
   S702_BT_CODE_2112.TEST_TEMP[8] := B#16#0;
   S702_BT_CODE_2112.TEST_TEMP[9] := B#16#0;
   S702_BT_CODE_2112.TEST_TEMP[10] := B#16#0;
   S702_BT_CODE_2112.TEST_TEMP[11] := B#16#0;
   S702_BT_CODE_2112.TEST_TEMP[12] := B#16#0;
   S702_BT_CODE_2112.TEST_TEMP[13] := B#16#0;
   S702_BT_CODE_2112.TEST_TEMP[14] := B#16#0;
   S702_BT_CODE_2112.TEST_TEMP[15] := B#16#0;
   S702_BT_CODE_2112.TEST_TEMP[16] := B#16#0;
   S702_BT_CODE_2112.TEST_TEMP[17] := B#16#0;
   S702_BT_CODE_2112.TEST_TEMP[18] := B#16#0;
   S702_BT_CODE_2112.TEST_TEMP[19] := B#16#0;
   S702_BT_CODE_2112.TEST_TEMP[20] := B#16#0;
   S702_BT_CODE_2112.TEST_TEMP[21] := B#16#0;
   S702_BT_CODE_2112.TEST_TEMP[22] := B#16#0;
   S702_BT_CODE_2112.TEST_TEMP[23] := B#16#0;
   S702_BT_CODE_2112.TEST_TEMP[24] := B#16#0;
   S702_BT_CODE_2112.TEST_TEMP[25] := B#16#0;
   S702_BT_CODE_2112.TEST_TEMP[26] := B#16#0;
   S702_BT_CODE_2112.TEST_TEMP[27] := B#16#0;
   S702_BT_CODE_2112.TEST_TEMP[28] := B#16#0;
   S702_BT_CODE_2112.TEST_TEMP[29] := B#16#0;
   S702_BT_CODE_2112.TEST_TEMP[30] := B#16#0;
   S702_BT_CODE_2112.TEST_TEMP[31] := B#16#0;
   S702_BT_CODE_2112.TEST_TEMP[32] := B#16#0;
   S702_BT_CODE_2112.TEST_TEMP[33] := B#16#0;
   S702_BT_CODE_2112.TEST_TEMP[34] := B#16#0;
   S702_BT_CODE_2112.TEST_TEMP[35] := B#16#0;
   S702_BT_CODE_2112.TEST_TEMP[36] := B#16#0;
   S702_BT_CODE_2112.TEST_TEMP[37] := B#16#0;
   S702_BT_CODE_2112.TEST_TEMP[38] := B#16#0;
   S702_BT_CODE_2112.TEST_TEMP[39] := B#16#0;
   S702_BT_CODE_2112.TEST_TEMP[40] := B#16#0;
   S702_BT_CODE_2113.STATION_MAIN := W#16#0;
   S702_BT_CODE_2113.DISTINCTION_LH_RH := W#16#0;
   S702_BT_CODE_2113.STAION_NUMBER := W#16#0;
   S702_BT_CODE_2113.BODY_TYPE_1ST := W#16#0;
   S702_BT_CODE_2113.BODY_TYPE_OPTION := W#16#0;
   S702_BT_CODE_2113.RBT1_STANDARD_WELD_DATA := W#16#0;
   S702_BT_CODE_2113.RBT2_STANDARD_WELD_DATA := W#16#0;
   S702_BT_CODE_2113.RBT3_STANDARD_WELD_DATA := W#16#0;
   S702_BT_CODE_2113.RBT4_STANDARD_WELD_DATA := W#16#0;
   S702_BT_CODE_2113.RBT5_STANDARD_WELD_DATA := W#16#0;
   S702_BT_CODE_2113.RBT6_STANDARD_WELD_DATA := W#16#0;
   S702_BT_CODE_2113.RBT7_STANDARD_WELD_DATA := W#16#0;
   S702_BT_CODE_2113.RBT8_STANDARD_WELD_DATA := W#16#0;
   S702_BT_CODE_2113.RBT9_STANDARD_WELD_DATA := W#16#0;
   S702_BT_CODE_2113.RBT10_STANDARD_WELD_DATA := W#16#0;
   S702_BT_CODE_2113.RBT11_STANDARD_WELD_DATA := W#16#0;
   S702_BT_CODE_2113.RBT12_STANDARD_WELD_DATA := W#16#0;
   S702_BT_CODE_2113.RBT13_STANDARD_WELD_DATA := W#16#0;
   S702_BT_CODE_2113.RBT14_STANDARD_WELD_DATA := W#16#0;
   S702_BT_CODE_2113.RBT15_STANDARD_WELD_DATA := W#16#0;
   S702_BT_CODE_2113.RBT16_STANDARD_WELD_DATA := W#16#0;
   S702_BT_CODE_2113.RBT17_STANDARD_WELD_DATA := W#16#0;
   S702_BT_CODE_2113.RBT18_STANDARD_WELD_DATA := W#16#0;
   S702_BT_CODE_2113.RBT19_STANDARD_WELD_DATA := W#16#0;
   S702_BT_CODE_2113.RBT20_STANDARD_WELD_DATA := W#16#0;
   S702_BT_CODE_2113.RBT21_STANDARD_WELD_DATA := W#16#0;
   S702_BT_CODE_2113.RBT22_STANDARD_WELD_DATA := W#16#0;
   S702_BT_CODE_2113.RBT23_STANDARD_WELD_DAT := W#16#0;
   S702_BT_CODE_2113.RBT24_STANDARD_WELD_DAT := W#16#0;
   S702_BT_CODE_2113.CHK_WORD := W#16#0;
   S702_BT_CODE_2113.TEST_TEMP[1] := B#16#0;
   S702_BT_CODE_2113.TEST_TEMP[2] := B#16#0;
   S702_BT_CODE_2113.TEST_TEMP[3] := B#16#0;
   S702_BT_CODE_2113.TEST_TEMP[4] := B#16#0;
   S702_BT_CODE_2113.TEST_TEMP[5] := B#16#0;
   S702_BT_CODE_2113.TEST_TEMP[6] := B#16#0;
   S702_BT_CODE_2113.TEST_TEMP[7] := B#16#0;
   S702_BT_CODE_2113.TEST_TEMP[8] := B#16#0;
   S702_BT_CODE_2113.TEST_TEMP[9] := B#16#0;
   S702_BT_CODE_2113.TEST_TEMP[10] := B#16#0;
   S702_BT_CODE_2113.TEST_TEMP[11] := B#16#0;
   S702_BT_CODE_2113.TEST_TEMP[12] := B#16#0;
   S702_BT_CODE_2113.TEST_TEMP[13] := B#16#0;
   S702_BT_CODE_2113.TEST_TEMP[14] := B#16#0;
   S702_BT_CODE_2113.TEST_TEMP[15] := B#16#0;
   S702_BT_CODE_2113.TEST_TEMP[16] := B#16#0;
   S702_BT_CODE_2113.TEST_TEMP[17] := B#16#0;
   S702_BT_CODE_2113.TEST_TEMP[18] := B#16#0;
   S702_BT_CODE_2113.TEST_TEMP[19] := B#16#0;
   S702_BT_CODE_2113.TEST_TEMP[20] := B#16#0;
   S702_BT_CODE_2113.TEST_TEMP[21] := B#16#0;
   S702_BT_CODE_2113.TEST_TEMP[22] := B#16#0;
   S702_BT_CODE_2113.TEST_TEMP[23] := B#16#0;
   S702_BT_CODE_2113.TEST_TEMP[24] := B#16#0;
   S702_BT_CODE_2113.TEST_TEMP[25] := B#16#0;
   S702_BT_CODE_2113.TEST_TEMP[26] := B#16#0;
   S702_BT_CODE_2113.TEST_TEMP[27] := B#16#0;
   S702_BT_CODE_2113.TEST_TEMP[28] := B#16#0;
   S702_BT_CODE_2113.TEST_TEMP[29] := B#16#0;
   S702_BT_CODE_2113.TEST_TEMP[30] := B#16#0;
   S702_BT_CODE_2113.TEST_TEMP[31] := B#16#0;
   S702_BT_CODE_2113.TEST_TEMP[32] := B#16#0;
   S702_BT_CODE_2113.TEST_TEMP[33] := B#16#0;
   S702_BT_CODE_2113.TEST_TEMP[34] := B#16#0;
   S702_BT_CODE_2113.TEST_TEMP[35] := B#16#0;
   S702_BT_CODE_2113.TEST_TEMP[36] := B#16#0;
   S702_BT_CODE_2113.TEST_TEMP[37] := B#16#0;
   S702_BT_CODE_2113.TEST_TEMP[38] := B#16#0;
   S702_BT_CODE_2113.TEST_TEMP[39] := B#16#0;
   S702_BT_CODE_2113.TEST_TEMP[40] := B#16#0;
   S702_BT_CODE_2114.STATION_MAIN := W#16#0;
   S702_BT_CODE_2114.DISTINCTION_LH_RH := W#16#0;
   S702_BT_CODE_2114.STAION_NUMBER := W#16#0;
   S702_BT_CODE_2114.BODY_TYPE_1ST := W#16#0;
   S702_BT_CODE_2114.BODY_TYPE_OPTION := W#16#0;
   S702_BT_CODE_2114.RBT1_STANDARD_WELD_DATA := W#16#0;
   S702_BT_CODE_2114.RBT2_STANDARD_WELD_DATA := W#16#0;
   S702_BT_CODE_2114.RBT3_STANDARD_WELD_DATA := W#16#0;
   S702_BT_CODE_2114.RBT4_STANDARD_WELD_DATA := W#16#0;
   S702_BT_CODE_2114.RBT5_STANDARD_WELD_DATA := W#16#0;
   S702_BT_CODE_2114.RBT6_STANDARD_WELD_DATA := W#16#0;
   S702_BT_CODE_2114.RBT7_STANDARD_WELD_DATA := W#16#0;
   S702_BT_CODE_2114.RBT8_STANDARD_WELD_DATA := W#16#0;
   S702_BT_CODE_2114.RBT9_STANDARD_WELD_DATA := W#16#0;
   S702_BT_CODE_2114.RBT10_STANDARD_WELD_DATA := W#16#0;
   S702_BT_CODE_2114.RBT11_STANDARD_WELD_DATA := W#16#0;
   S702_BT_CODE_2114.RBT12_STANDARD_WELD_DATA := W#16#0;
   S702_BT_CODE_2114.RBT13_STANDARD_WELD_DATA := W#16#0;
   S702_BT_CODE_2114.RBT14_STANDARD_WELD_DATA := W#16#0;
   S702_BT_CODE_2114.RBT15_STANDARD_WELD_DATA := W#16#0;
   S702_BT_CODE_2114.RBT16_STANDARD_WELD_DATA := W#16#0;
   S702_BT_CODE_2114.RBT17_STANDARD_WELD_DATA := W#16#0;
   S702_BT_CODE_2114.RBT18_STANDARD_WELD_DATA := W#16#0;
   S702_BT_CODE_2114.RBT19_STANDARD_WELD_DATA := W#16#0;
   S702_BT_CODE_2114.RBT20_STANDARD_WELD_DATA := W#16#0;
   S702_BT_CODE_2114.RBT21_STANDARD_WELD_DATA := W#16#0;
   S702_BT_CODE_2114.RBT22_STANDARD_WELD_DATA := W#16#0;
   S702_BT_CODE_2114.RBT23_STANDARD_WELD_DAT := W#16#0;
   S702_BT_CODE_2114.RBT24_STANDARD_WELD_DAT := W#16#0;
   S702_BT_CODE_2114.CHK_WORD := W#16#0;
   S702_BT_CODE_2114.TEST_TEMP[1] := B#16#0;
   S702_BT_CODE_2114.TEST_TEMP[2] := B#16#0;
   S702_BT_CODE_2114.TEST_TEMP[3] := B#16#0;
   S702_BT_CODE_2114.TEST_TEMP[4] := B#16#0;
   S702_BT_CODE_2114.TEST_TEMP[5] := B#16#0;
   S702_BT_CODE_2114.TEST_TEMP[6] := B#16#0;
   S702_BT_CODE_2114.TEST_TEMP[7] := B#16#0;
   S702_BT_CODE_2114.TEST_TEMP[8] := B#16#0;
   S702_BT_CODE_2114.TEST_TEMP[9] := B#16#0;
   S702_BT_CODE_2114.TEST_TEMP[10] := B#16#0;
   S702_BT_CODE_2114.TEST_TEMP[11] := B#16#0;
   S702_BT_CODE_2114.TEST_TEMP[12] := B#16#0;
   S702_BT_CODE_2114.TEST_TEMP[13] := B#16#0;
   S702_BT_CODE_2114.TEST_TEMP[14] := B#16#0;
   S702_BT_CODE_2114.TEST_TEMP[15] := B#16#0;
   S702_BT_CODE_2114.TEST_TEMP[16] := B#16#0;
   S702_BT_CODE_2114.TEST_TEMP[17] := B#16#0;
   S702_BT_CODE_2114.TEST_TEMP[18] := B#16#0;
   S702_BT_CODE_2114.TEST_TEMP[19] := B#16#0;
   S702_BT_CODE_2114.TEST_TEMP[20] := B#16#0;
   S702_BT_CODE_2114.TEST_TEMP[21] := B#16#0;
   S702_BT_CODE_2114.TEST_TEMP[22] := B#16#0;
   S702_BT_CODE_2114.TEST_TEMP[23] := B#16#0;
   S702_BT_CODE_2114.TEST_TEMP[24] := B#16#0;
   S702_BT_CODE_2114.TEST_TEMP[25] := B#16#0;
   S702_BT_CODE_2114.TEST_TEMP[26] := B#16#0;
   S702_BT_CODE_2114.TEST_TEMP[27] := B#16#0;
   S702_BT_CODE_2114.TEST_TEMP[28] := B#16#0;
   S702_BT_CODE_2114.TEST_TEMP[29] := B#16#0;
   S702_BT_CODE_2114.TEST_TEMP[30] := B#16#0;
   S702_BT_CODE_2114.TEST_TEMP[31] := B#16#0;
   S702_BT_CODE_2114.TEST_TEMP[32] := B#16#0;
   S702_BT_CODE_2114.TEST_TEMP[33] := B#16#0;
   S702_BT_CODE_2114.TEST_TEMP[34] := B#16#0;
   S702_BT_CODE_2114.TEST_TEMP[35] := B#16#0;
   S702_BT_CODE_2114.TEST_TEMP[36] := B#16#0;
   S702_BT_CODE_2114.TEST_TEMP[37] := B#16#0;
   S702_BT_CODE_2114.TEST_TEMP[38] := B#16#0;
   S702_BT_CODE_2114.TEST_TEMP[39] := B#16#0;
   S702_BT_CODE_2114.TEST_TEMP[40] := B#16#0;
   S702_BT_CODE_2115.STATION_MAIN := W#16#0;
   S702_BT_CODE_2115.DISTINCTION_LH_RH := W#16#0;
   S702_BT_CODE_2115.STAION_NUMBER := W#16#0;
   S702_BT_CODE_2115.BODY_TYPE_1ST := W#16#0;
   S702_BT_CODE_2115.BODY_TYPE_OPTION := W#16#0;
   S702_BT_CODE_2115.RBT1_STANDARD_WELD_DATA := W#16#0;
   S702_BT_CODE_2115.RBT2_STANDARD_WELD_DATA := W#16#0;
   S702_BT_CODE_2115.RBT3_STANDARD_WELD_DATA := W#16#0;
   S702_BT_CODE_2115.RBT4_STANDARD_WELD_DATA := W#16#0;
   S702_BT_CODE_2115.RBT5_STANDARD_WELD_DATA := W#16#0;
   S702_BT_CODE_2115.RBT6_STANDARD_WELD_DATA := W#16#0;
   S702_BT_CODE_2115.RBT7_STANDARD_WELD_DATA := W#16#0;
   S702_BT_CODE_2115.RBT8_STANDARD_WELD_DATA := W#16#0;
   S702_BT_CODE_2115.RBT9_STANDARD_WELD_DATA := W#16#0;
   S702_BT_CODE_2115.RBT10_STANDARD_WELD_DATA := W#16#0;
   S702_BT_CODE_2115.RBT11_STANDARD_WELD_DATA := W#16#0;
   S702_BT_CODE_2115.RBT12_STANDARD_WELD_DATA := W#16#0;
   S702_BT_CODE_2115.RBT13_STANDARD_WELD_DATA := W#16#0;
   S702_BT_CODE_2115.RBT14_STANDARD_WELD_DATA := W#16#0;
   S702_BT_CODE_2115.RBT15_STANDARD_WELD_DATA := W#16#0;
   S702_BT_CODE_2115.RBT16_STANDARD_WELD_DATA := W#16#0;
   S702_BT_CODE_2115.RBT17_STANDARD_WELD_DATA := W#16#0;
   S702_BT_CODE_2115.RBT18_STANDARD_WELD_DATA := W#16#0;
   S702_BT_CODE_2115.RBT19_STANDARD_WELD_DATA := W#16#0;
   S702_BT_CODE_2115.RBT20_STANDARD_WELD_DATA := W#16#0;
   S702_BT_CODE_2115.RBT21_STANDARD_WELD_DATA := W#16#0;
   S702_BT_CODE_2115.RBT22_STANDARD_WELD_DATA := W#16#0;
   S702_BT_CODE_2115.RBT23_STANDARD_WELD_DAT := W#16#0;
   S702_BT_CODE_2115.RBT24_STANDARD_WELD_DAT := W#16#0;
   S702_BT_CODE_2115.CHK_WORD := W#16#0;
   S702_BT_CODE_2115.TEST_TEMP[1] := B#16#0;
   S702_BT_CODE_2115.TEST_TEMP[2] := B#16#0;
   S702_BT_CODE_2115.TEST_TEMP[3] := B#16#0;
   S702_BT_CODE_2115.TEST_TEMP[4] := B#16#0;
   S702_BT_CODE_2115.TEST_TEMP[5] := B#16#0;
   S702_BT_CODE_2115.TEST_TEMP[6] := B#16#0;
   S702_BT_CODE_2115.TEST_TEMP[7] := B#16#0;
   S702_BT_CODE_2115.TEST_TEMP[8] := B#16#0;
   S702_BT_CODE_2115.TEST_TEMP[9] := B#16#0;
   S702_BT_CODE_2115.TEST_TEMP[10] := B#16#0;
   S702_BT_CODE_2115.TEST_TEMP[11] := B#16#0;
   S702_BT_CODE_2115.TEST_TEMP[12] := B#16#0;
   S702_BT_CODE_2115.TEST_TEMP[13] := B#16#0;
   S702_BT_CODE_2115.TEST_TEMP[14] := B#16#0;
   S702_BT_CODE_2115.TEST_TEMP[15] := B#16#0;
   S702_BT_CODE_2115.TEST_TEMP[16] := B#16#0;
   S702_BT_CODE_2115.TEST_TEMP[17] := B#16#0;
   S702_BT_CODE_2115.TEST_TEMP[18] := B#16#0;
   S702_BT_CODE_2115.TEST_TEMP[19] := B#16#0;
   S702_BT_CODE_2115.TEST_TEMP[20] := B#16#0;
   S702_BT_CODE_2115.TEST_TEMP[21] := B#16#0;
   S702_BT_CODE_2115.TEST_TEMP[22] := B#16#0;
   S702_BT_CODE_2115.TEST_TEMP[23] := B#16#0;
   S702_BT_CODE_2115.TEST_TEMP[24] := B#16#0;
   S702_BT_CODE_2115.TEST_TEMP[25] := B#16#0;
   S702_BT_CODE_2115.TEST_TEMP[26] := B#16#0;
   S702_BT_CODE_2115.TEST_TEMP[27] := B#16#0;
   S702_BT_CODE_2115.TEST_TEMP[28] := B#16#0;
   S702_BT_CODE_2115.TEST_TEMP[29] := B#16#0;
   S702_BT_CODE_2115.TEST_TEMP[30] := B#16#0;
   S702_BT_CODE_2115.TEST_TEMP[31] := B#16#0;
   S702_BT_CODE_2115.TEST_TEMP[32] := B#16#0;
   S702_BT_CODE_2115.TEST_TEMP[33] := B#16#0;
   S702_BT_CODE_2115.TEST_TEMP[34] := B#16#0;
   S702_BT_CODE_2115.TEST_TEMP[35] := B#16#0;
   S702_BT_CODE_2115.TEST_TEMP[36] := B#16#0;
   S702_BT_CODE_2115.TEST_TEMP[37] := B#16#0;
   S702_BT_CODE_2115.TEST_TEMP[38] := B#16#0;
   S702_BT_CODE_2115.TEST_TEMP[39] := B#16#0;
   S702_BT_CODE_2115.TEST_TEMP[40] := B#16#0;
   S702_BT_CODE_2116.STATION_MAIN := W#16#0;
   S702_BT_CODE_2116.DISTINCTION_LH_RH := W#16#0;
   S702_BT_CODE_2116.STAION_NUMBER := W#16#0;
   S702_BT_CODE_2116.BODY_TYPE_1ST := W#16#0;
   S702_BT_CODE_2116.BODY_TYPE_OPTION := W#16#0;
   S702_BT_CODE_2116.RBT1_STANDARD_WELD_DATA := W#16#0;
   S702_BT_CODE_2116.RBT2_STANDARD_WELD_DATA := W#16#0;
   S702_BT_CODE_2116.RBT3_STANDARD_WELD_DATA := W#16#0;
   S702_BT_CODE_2116.RBT4_STANDARD_WELD_DATA := W#16#0;
   S702_BT_CODE_2116.RBT5_STANDARD_WELD_DATA := W#16#0;
   S702_BT_CODE_2116.RBT6_STANDARD_WELD_DATA := W#16#0;
   S702_BT_CODE_2116.RBT7_STANDARD_WELD_DATA := W#16#0;
   S702_BT_CODE_2116.RBT8_STANDARD_WELD_DATA := W#16#0;
   S702_BT_CODE_2116.RBT9_STANDARD_WELD_DATA := W#16#0;
   S702_BT_CODE_2116.RBT10_STANDARD_WELD_DATA := W#16#0;
   S702_BT_CODE_2116.RBT11_STANDARD_WELD_DATA := W#16#0;
   S702_BT_CODE_2116.RBT12_STANDARD_WELD_DATA := W#16#0;
   S702_BT_CODE_2116.RBT13_STANDARD_WELD_DATA := W#16#0;
   S702_BT_CODE_2116.RBT14_STANDARD_WELD_DATA := W#16#0;
   S702_BT_CODE_2116.RBT15_STANDARD_WELD_DATA := W#16#0;
   S702_BT_CODE_2116.RBT16_STANDARD_WELD_DATA := W#16#0;
   S702_BT_CODE_2116.RBT17_STANDARD_WELD_DATA := W#16#0;
   S702_BT_CODE_2116.RBT18_STANDARD_WELD_DATA := W#16#0;
   S702_BT_CODE_2116.RBT19_STANDARD_WELD_DATA := W#16#0;
   S702_BT_CODE_2116.RBT20_STANDARD_WELD_DATA := W#16#0;
   S702_BT_CODE_2116.RBT21_STANDARD_WELD_DATA := W#16#0;
   S702_BT_CODE_2116.RBT22_STANDARD_WELD_DATA := W#16#0;
   S702_BT_CODE_2116.RBT23_STANDARD_WELD_DAT := W#16#0;
   S702_BT_CODE_2116.RBT24_STANDARD_WELD_DAT := W#16#0;
   S702_BT_CODE_2116.CHK_WORD := W#16#0;
   S702_BT_CODE_2116.TEST_TEMP[1] := B#16#0;
   S702_BT_CODE_2116.TEST_TEMP[2] := B#16#0;
   S702_BT_CODE_2116.TEST_TEMP[3] := B#16#0;
   S702_BT_CODE_2116.TEST_TEMP[4] := B#16#0;
   S702_BT_CODE_2116.TEST_TEMP[5] := B#16#0;
   S702_BT_CODE_2116.TEST_TEMP[6] := B#16#0;
   S702_BT_CODE_2116.TEST_TEMP[7] := B#16#0;
   S702_BT_CODE_2116.TEST_TEMP[8] := B#16#0;
   S702_BT_CODE_2116.TEST_TEMP[9] := B#16#0;
   S702_BT_CODE_2116.TEST_TEMP[10] := B#16#0;
   S702_BT_CODE_2116.TEST_TEMP[11] := B#16#0;
   S702_BT_CODE_2116.TEST_TEMP[12] := B#16#0;
   S702_BT_CODE_2116.TEST_TEMP[13] := B#16#0;
   S702_BT_CODE_2116.TEST_TEMP[14] := B#16#0;
   S702_BT_CODE_2116.TEST_TEMP[15] := B#16#0;
   S702_BT_CODE_2116.TEST_TEMP[16] := B#16#0;
   S702_BT_CODE_2116.TEST_TEMP[17] := B#16#0;
   S702_BT_CODE_2116.TEST_TEMP[18] := B#16#0;
   S702_BT_CODE_2116.TEST_TEMP[19] := B#16#0;
   S702_BT_CODE_2116.TEST_TEMP[20] := B#16#0;
   S702_BT_CODE_2116.TEST_TEMP[21] := B#16#0;
   S702_BT_CODE_2116.TEST_TEMP[22] := B#16#0;
   S702_BT_CODE_2116.TEST_TEMP[23] := B#16#0;
   S702_BT_CODE_2116.TEST_TEMP[24] := B#16#0;
   S702_BT_CODE_2116.TEST_TEMP[25] := B#16#0;
   S702_BT_CODE_2116.TEST_TEMP[26] := B#16#0;
   S702_BT_CODE_2116.TEST_TEMP[27] := B#16#0;
   S702_BT_CODE_2116.TEST_TEMP[28] := B#16#0;
   S702_BT_CODE_2116.TEST_TEMP[29] := B#16#0;
   S702_BT_CODE_2116.TEST_TEMP[30] := B#16#0;
   S702_BT_CODE_2116.TEST_TEMP[31] := B#16#0;
   S702_BT_CODE_2116.TEST_TEMP[32] := B#16#0;
   S702_BT_CODE_2116.TEST_TEMP[33] := B#16#0;
   S702_BT_CODE_2116.TEST_TEMP[34] := B#16#0;
   S702_BT_CODE_2116.TEST_TEMP[35] := B#16#0;
   S702_BT_CODE_2116.TEST_TEMP[36] := B#16#0;
   S702_BT_CODE_2116.TEST_TEMP[37] := B#16#0;
   S702_BT_CODE_2116.TEST_TEMP[38] := B#16#0;
   S702_BT_CODE_2116.TEST_TEMP[39] := B#16#0;
   S702_BT_CODE_2116.TEST_TEMP[40] := B#16#0;
   S702_BT_CODE_2117.STATION_MAIN := W#16#0;
   S702_BT_CODE_2117.DISTINCTION_LH_RH := W#16#0;
   S702_BT_CODE_2117.STAION_NUMBER := W#16#0;
   S702_BT_CODE_2117.BODY_TYPE_1ST := W#16#0;
   S702_BT_CODE_2117.BODY_TYPE_OPTION := W#16#0;
   S702_BT_CODE_2117.RBT1_STANDARD_WELD_DATA := W#16#0;
   S702_BT_CODE_2117.RBT2_STANDARD_WELD_DATA := W#16#0;
   S702_BT_CODE_2117.RBT3_STANDARD_WELD_DATA := W#16#0;
   S702_BT_CODE_2117.RBT4_STANDARD_WELD_DATA := W#16#0;
